KUKA KRL program: EPS_2_25694_RR01_A_20260120031656.src

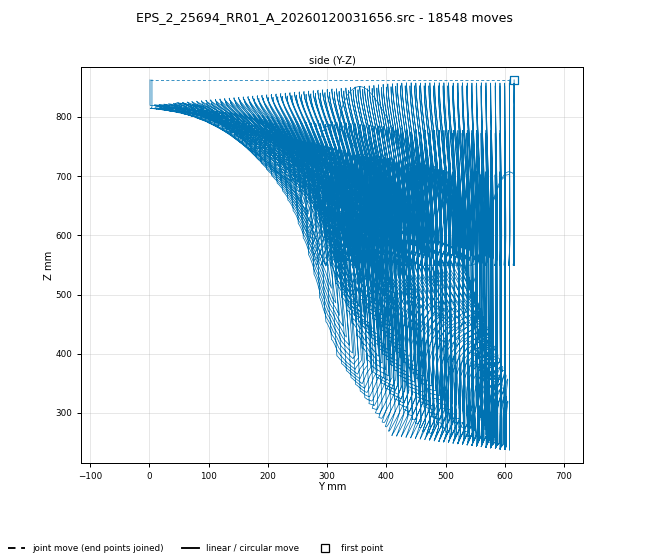
[picture p0: tool path of EPS_2_25694_RR01_A_20260120031656.src, 18548 of 18550 moves have a stored position in this frame; points joined in program order, loops and branches not executed]
&ACCESS RVP
&REL 4
&COMMENT QRS 19112012
&PARAM EDITMASK = *
DEF PART()
EXT BAS (BAS_COMMAND :IN,REAL :IN )
INT I
BAS (#INITMOV,0 )

;KUKA QRS Post kuka4.cps  Date:22-06-2017 !

File_ID=2993

QRS_PRE_INIT()

;Init var - Until changes are made in qrs_pre_init
Outlet_Square_prg=0
Inlet_1_Square_prg=0
Inlet_2_Square_prg=0
Inlet_3_Square_prg=0
Inlet_4_Square_prg=0
Inlet_5_Square_prg=0

Outlet_1={X 0.000, Y 425.000, Z 586.000, B 0.000, E1 0.000 }
Inlet_1={X 0.000, Y 537.740, Z 427.000, B 0.000, E1 94.000 }
Inlet_2={X 0.000, Y 466.000, Z 544.000, B 0.000, E1 177.000 }
Inlet_3={X 0.000, Y 531.490, Z 452.000, B 0.000, E1 275.000 }
Outlet_1_type=533
Inlet_1_type=201
Inlet_2_type=457
Inlet_3_type=251
;QRS#1=Sidecore dimensions
;QRS#2=525-21" Concrete
;QRS#3=200-8" PVC SDR 35
;QRS#4=450-18" Concrete
;QRS#5=250-10" PVC SDR 35
;QRS#6=
;QRS#7=
;QRS#8=
;QRS#9=S306-32
;QRS#10=12-08 PSX
;QRS#11=28A PSX-2
;QRS#12=14M PSX
;QRS#13=
;QRS#14=
;QRS#15=
;QRS#16=1220x127x1219 4'
;QRS#17=EPS Height
;QRS#18=852,5
;QRS#19=*
;QRS#20= UPDATED VERSION 22-06-2017
;QRS#21=*
Outlet_Square=0250
Inlet_1_Square=0100
Inlet_2_Square=0250
Inlet_3_Square=0100
Inlet_4_Square=0
Inlet_5_Square=0
Mill_Square=1
Outlet_Square_Prg=263
Inlet_1_Square_prg=204
Inlet_2_Square_prg=274
Inlet_3_Square_prg=205

QRS_INIT()

$ADVANCE=5

; T1
PTP {E1 172.342,E2 172.342}
PTP {X 0,Y 615.793,A -85,B 0,C 180,E1 172.342,E2 172.342,E3 0,E4 0,E5 0,E6 0}
QRS_SPEED_INIT()
LIN {X 0,Y 615.793,Z 862.5,A -85,B 0,C 180,E1 172.342,E2 172.342,E3 0,E4 0,E5 0,E6 0} C_VEL
LIN {X 0,Y 615.793,Z 711.666,A -85,B 0,C 180,E1 172.342,E2 172.342} C_VEL
LIN {X 0,Y 615.793,Z 703.764,A -85,B 0,C 180,E1 172.342,E2 172.342} C_VEL
LIN {X 0,Y 615.77,Z 701.828,A -85,B 0,C 180,E1 172.575,E2 172.575} C_VEL
LIN {X 0,Y 615.76,Z 703.691,A -85,B 0,C 180,E1 173.245,E2 173.245} C_VEL
LIN {X 0,Y 615.844,Z 705.541,A -85,B 0,C 180,E1 174.193,E2 174.193} C_VEL
LIN {X 0,Y 615.719,Z 706.621,A -85,B 0,C 180,E1 175.124,E2 175.124} C_VEL
LIN {X 0,Y 615.715,Z 706.871,A -85,B 0,C 180,E1 175.589,E2 175.589} C_VEL
LIN {X 0,Y 615.813,Z 706.79,A -85,B 0,C 180,E1 176.52,E2 176.52} C_VEL
LIN {X 0,Y 615.76,Z 705.947,A -85,B 0,C 180,E1 177.448,E2 177.448} C_VEL
LIN {X 0,Y 615.722,Z 704.334,A -85,B 0,C 180,E1 178.376,E2 178.376} C_VEL
LIN {X 0,Y 615.846,Z 701.911,A -85,B 0,C 180,E1 179.304,E2 179.304} C_VEL
LIN {X 0,Y 615.823,Z 700.411,A -85,B 0,C 180,E1 179.768,E2 179.768} C_VEL
LIN {X 0,Y 615.774,Z 698.687,A -85,B 0,C 180,E1 180.232,E2 180.232} C_VEL
LIN {X 0,Y 615.76,Z 695.634,A -85,B 0,C 180,E1 180.928,E2 180.928} C_VEL
LIN {X 0,Y 615.848,Z 692.021,A -85,B 0,C 180,E1 181.623,E2 181.623} C_VEL
LIN {X 0,Y 615.81,Z 687.854,A -85,B 0,C 180,E1 182.319,E2 182.319} C_VEL
LIN {X 0,Y 615.8,Z 682.955,A -85,B 0,C 180,E1 183.016,E2 183.016} C_VEL
LIN {X 0,Y 615.841,Z 677.301,A -85,B 0,C 180,E1 183.713,E2 183.713} C_VEL
LIN {X 0,Y 615.831,Z 671.884,A -85,B 0,C 180,E1 184.294,E2 184.294} C_VEL
LIN {X 0,Y 615.826,Z 665.734,A -85,B 0,C 180,E1 184.875,E2 184.875} C_VEL
LIN {X 0,Y 615.847,Z 658.636,A -85,B 0,C 180,E1 185.457,E2 185.457} C_VEL
LIN {X 0,Y 615.854,Z 652.201,A -85,B 0,C 180,E1 185.918,E2 185.918} C_VEL
LIN {X 0,Y 615.823,Z 645.096,A -85,B 0,C 180,E1 186.362,E2 186.362} C_VEL
LIN {X 0,Y 615.837,Z 636.811,A -85,B 0,C 180,E1 186.805,E2 186.805} C_VEL
LIN {X 0,Y 615.843,Z 629.456,A -85,B 0,C 180,E1 187.138,E2 187.138} C_VEL
LIN {X 0,Y 615.852,Z 620.279,A -85,B 0,C 180,E1 187.484,E2 187.484} C_VEL
LIN {X 0,Y 615.848,Z 611.384,A -85,B 0,C 180,E1 187.748,E2 187.748} C_VEL
LIN {X 0,Y 615.849,Z 602.82,A -85,B 0,C 180,E1 187.941,E2 187.941} C_VEL
LIN {X 0,Y 615.85,Z 593.381,A -85,B 0,C 180,E1 188.09,E2 188.09} C_VEL
LIN {X 0,Y 615.685,Z 559.528,A -85,B 0,C 180,E1 188.49,E2 188.49} C_VEL
LIN {X 0,Y 615.331,Z 549.53,A -85,B 0,C 180,E1 188.614,E2 188.614} C_VEL
LIN {X 0,Y 615.64,Z 549.53,A -85,B 0,C 180,E1 188.676,E2 188.676} C_VEL
LIN {X 0,Y 615.827,Z 549.53,A -85,B 0,C 180,E1 189.302,E2 189.302} C_VEL
LIN {X 0,Y 615.855,Z 549.53,A -85,B 0,C 180,E1 190.493,E2 190.493} C_VEL
LIN {X 0,Y 615.807,Z 549.53,A -85,B 0,C 180,E1 195.252,E2 195.252} C_VEL
LIN {X 0,Y 615.774,Z 549.53,A -85,B 0,C 180,E1 200.122,E2 200.122} C_VEL
LIN {X 0,Y 615.735,Z 549.53,A -85,B 0,C 180,E1 205.151,E2 205.151} C_VEL
LIN {X 0,Y 615.403,Z 549.53,A -85,B 0,C 180,E1 209.459,E2 209.459} C_VEL
LIN {X 0,Y 615.737,Z 549.53,A -85,B 0,C 180,E1 210.395,E2 210.395} C_VEL
LIN {X 0,Y 615.132,Z 549.53,A -85,B 0,C 180,E1 213.842,E2 213.842} C_VEL
LIN {X 0,Y 615.665,Z 549.53,A -85,B 0,C 180,E1 215.943,E2 215.943} C_VEL
LIN {X 0,Y 615.412,Z 549.53,A -85,B 0,C 180,E1 217.842,E2 217.842} C_VEL
LIN {X 0,Y 615.369,Z 549.53,A -85,B 0,C 180,E1 218.885,E2 218.885} C_VEL
LIN {X 0,Y 615.653,Z 549.53,A -85,B 0,C 180,E1 221.504,E2 221.504} C_VEL
LIN {X 0,Y 615.675,Z 549.53,A -85,B 0,C 180,E1 225.105,E2 225.105} C_VEL
LIN {X 0,Y 615.271,Z 549.53,A -85,B 0,C 180,E1 228.537,E2 228.537} C_VEL
LIN {X 0,Y 615.658,Z 549.53,A -85,B 0,C 180,E1 231.137,E2 231.137} C_VEL
LIN {X 0,Y 615.637,Z 549.53,A -85,B 0,C 180,E1 236.088,E2 236.088} C_VEL
LIN {X 0,Y 615.75,Z 549.53,A -85,B 0,C 180,E1 236.878,E2 236.878} C_VEL
LIN {X 0,Y 615.843,Z 549.53,A -85,B 0,C 180,E1 240.621,E2 240.621} C_VEL
LIN {X 0,Y 615.218,Z 549.53,A -85,B 0,C 180,E1 240.78,E2 240.78} C_VEL
LIN {X 0,Y 615.11,Z 550.038,A -85,B 0,C 180,E1 240.802,E2 240.802} C_VEL
LIN {X 0,Y 615.44,Z 600.029,A -85,B 0,C 180,E1 241.477,E2 241.477} C_VEL
LIN {X 0,Y 615.51,Z 611.094,A -85,B 0,C 180,E1 241.655,E2 241.655} C_VEL
LIN {X 0,Y 615.537,Z 625.6,A -85,B 0,C 180,E1 241.961,E2 241.961} C_VEL
LIN {X 0,Y 615.51,Z 635.908,A -85,B 0,C 180,E1 242.221,E2 242.221} C_VEL
LIN {X 0,Y 615.677,Z 651.509,A -85,B 0,C 180,E1 242.705,E2 242.705} C_VEL
LIN {X 0,Y 615.645,Z 663.945,A -85,B 0,C 180,E1 243.152,E2 243.152} C_VEL
LIN {X 0,Y 615.577,Z 673.861,A -85,B 0,C 180,E1 243.554,E2 243.554} C_VEL
LIN {X 0,Y 615.711,Z 689.587,A -85,B 0,C 180,E1 244.286,E2 244.286} C_VEL
LIN {X 0,Y 615.692,Z 701.936,A -85,B 0,C 180,E1 244.935,E2 244.935} C_VEL
LIN {X 0,Y 615.677,Z 713.616,A -85,B 0,C 180,E1 245.617,E2 245.617} C_VEL
LIN {X 0,Y 615.714,Z 725.406,A -85,B 0,C 180,E1 246.38,E2 246.38} C_VEL
LIN {X 0,Y 615.721,Z 736.083,A -85,B 0,C 180,E1 247.135,E2 247.135} C_VEL
LIN {X 0,Y 615.707,Z 747.387,A -85,B 0,C 180,E1 248.011,E2 248.011} C_VEL
LIN {X 0,Y 615.704,Z 756.649,A -85,B 0,C 180,E1 248.791,E2 248.791} C_VEL
LIN {X 0,Y 615.752,Z 766.786,A -85,B 0,C 180,E1 249.722,E2 249.722} C_VEL
LIN {X 0,Y 615.723,Z 776.05,A -85,B 0,C 180,E1 250.646,E2 250.646} C_VEL
LIN {X 0,Y 615.683,Z 784.412,A -85,B 0,C 180,E1 251.548,E2 251.548} C_VEL
LIN {X 0,Y 615.766,Z 792.772,A -85,B 0,C 180,E1 252.531,E2 252.531} C_VEL
LIN {X 0,Y 615.718,Z 800.678,A -85,B 0,C 180,E1 253.541,E2 253.541} C_VEL
LIN {X 0,Y 615.581,Z 807.424,A -85,B 0,C 180,E1 254.472,E2 254.472} C_VEL
LIN {X 0,Y 615.671,Z 815.058,A -85,B 0,C 180,E1 255.644,E2 255.644} C_VEL
LIN {X 0,Y 615.807,Z 820.435,A -85,B 0,C 180,E1 256.543,E2 256.543} C_VEL
LIN {X 0,Y 615.575,Z 826.908,A -85,B 0,C 180,E1 257.728,E2 257.728} C_VEL
LIN {X 0,Y 615.615,Z 832.623,A -85,B 0,C 180,E1 258.913,E2 258.913} C_VEL
LIN {X 0,Y 615.829,Z 837.633,A -85,B 0,C 180,E1 260.096,E2 260.096} C_VEL
LIN {X 0,Y 615.604,Z 842.062,A -85,B 0,C 180,E1 261.268,E2 261.268} C_VEL
LIN {X 0,Y 615.654,Z 846.465,A -85,B 0,C 180,E1 262.658,E2 262.658} C_VEL
LIN {X 0,Y 615.788,Z 849.368,A -85,B 0,C 180,E1 263.748,E2 263.748} C_VEL
LIN {X 0,Y 615.542,Z 852.381,A -85,B 0,C 180,E1 265.122,E2 265.122} C_VEL
LIN {X 0,Y 615.642,Z 854.591,A -85,B 0,C 180,E1 266.519,E2 266.519} C_VEL
LIN {X 0,Y 615.712,Z 856.054,A -85,B 0,C 180,E1 267.912,E2 267.912} C_VEL
LIN {X 0,Y 615.553,Z 856.715,A -85,B 0,C 180,E1 268.84,E2 268.84} C_VEL
LIN {X 0,Y 615.842,Z 856.659,A -85,B 0,C 180,E1 271.159,E2 271.159} C_VEL
LIN {X 0,Y 615.631,Z 856.069,A -85,B 0,C 180,E1 272.088,E2 272.088} C_VEL
LIN {X 0,Y 615.55,Z 854.608,A -85,B 0,C 180,E1 273.482,E2 273.482} C_VEL
LIN {X 0,Y 615.828,Z 852.329,A -85,B 0,C 180,E1 274.875,E2 274.875} C_VEL
LIN {X 0,Y 615.615,Z 849.404,A -85,B 0,C 180,E1 276.251,E2 276.251} C_VEL
LIN {X 0,Y 615.622,Z 846.266,A -85,B 0,C 180,E1 277.418,E2 277.418} C_VEL
LIN {X 0,Y 615.784,Z 842.035,A -85,B 0,C 180,E1 278.73,E2 278.73} C_VEL
LIN {X 0,Y 615.572,Z 837.67,A -85,B 0,C 180,E1 279.908,E2 279.908} C_VEL
LIN {X 0,Y 615.632,Z 832.621,A -85,B 0,C 180,E1 281.087,E2 281.087} C_VEL
LIN {X 0,Y 615.805,Z 826.881,A -85,B 0,C 180,E1 282.267,E2 282.267} C_VEL
LIN {X 0,Y 615.626,Z 820.453,A -85,B 0,C 180,E1 283.461,E2 283.461} C_VEL
LIN {X 0,Y 615.698,Z 813.192,A -85,B 0,C 180,E1 284.655,E2 284.655} C_VEL
LIN {X 0,Y 615.811,Z 807.63,A -85,B 0,C 180,E1 285.489,E2 285.489} C_VEL
LIN {X 0,Y 615.663,Z 798.196,A -85,B 0,C 180,E1 286.791,E2 286.791} C_VEL
LIN {X 0,Y 615.737,Z 789.604,A -85,B 0,C 180,E1 287.853,E2 287.853} C_VEL
LIN {X 0,Y 615.77,Z 781.409,A -85,B 0,C 180,E1 288.785,E2 288.785} C_VEL
LIN {X 0,Y 615.697,Z 771.52,A -85,B 0,C 180,E1 289.817,E2 289.817} C_VEL
LIN {X 0,Y 615.715,Z 763.533,A -85,B 0,C 180,E1 290.588,E2 290.588} C_VEL
LIN {X 0,Y 615.746,Z 753.03,A -85,B 0,C 180,E1 291.519,E2 291.519} C_VEL
LIN {X 0,Y 615.704,Z 743.049,A -85,B 0,C 180,E1 292.335,E2 292.335} C_VEL
LIN {X 0,Y 615.702,Z 733.289,A -85,B 0,C 180,E1 293.072,E2 293.072} C_VEL
LIN {X 0,Y 615.683,Z 721.63,A -85,B 0,C 180,E1 293.874,E2 293.874} C_VEL
LIN {X 0,Y 615.688,Z 709.594,A -85,B 0,C 180,E1 294.624,E2 294.624} C_VEL
LIN {X 0,Y 615.65,Z 698.88,A -85,B 0,C 180,E1 295.235,E2 295.235} C_VEL
LIN {X 0,Y 615.644,Z 688.01,A -85,B 0,C 180,E1 295.797,E2 295.797} C_VEL
LIN {X 0,Y 615.702,Z 673.863,A -85,B 0,C 180,E1 296.44,E2 296.44} C_VEL
LIN {X 0,Y 615.617,Z 660.66,A -85,B 0,C 180,E1 296.972,E2 296.972} C_VEL
LIN {X 0,Y 615.561,Z 651.512,A -85,B 0,C 180,E1 297.3,E2 297.3} C_VEL
LIN {X 0,Y 615.623,Z 634.838,A -85,B 0,C 180,E1 297.801,E2 297.801} C_VEL
LIN {X 0,Y 615.442,Z 622.423,A -85,B 0,C 180,E1 298.118,E2 298.118} C_VEL
LIN {X 0,Y 615.592,Z 610.944,A -85,B 0,C 180,E1 298.344,E2 298.344} C_VEL
LIN {X 0,Y 615.568,Z 593.456,A -85,B 0,C 180,E1 298.608,E2 298.608} C_VEL
LIN {X 0,Y 615.164,Z 549.53,A -85,B 0,C 180,E1 299.213,E2 299.213} C_VEL
LIN {X 0,Y 615.78,Z 549.53,A -85,B 0,C 180,E1 299.347,E2 299.347} C_VEL
LIN {X 0,Y 615.858,Z 549.53,A -85,B 0,C 180,E1 300.388,E2 300.388} C_VEL
LIN {X 0,Y 615.152,Z 549.53,A -85,B 0,C 180,E1 303.844,E2 303.844} C_VEL
LIN {X 0,Y 615.699,Z 549.53,A -85,B 0,C 180,E1 305.94,E2 305.94} C_VEL
LIN {X 0,Y 615.75,Z 549.53,A -85,B 0,C 180,E1 308.856,E2 308.856} C_VEL
LIN {X 0,Y 615.251,Z 549.53,A -85,B 0,C 180,E1 311.943,E2 311.943} C_VEL
LIN {X 0,Y 615.68,Z 549.53,A -85,B 0,C 180,E1 314.895,E2 314.895} C_VEL
LIN {X 0,Y 615.655,Z 549.53,A -85,B 0,C 180,E1 318.496,E2 318.496} C_VEL
LIN {X 0,Y 615.378,Z 549.53,A -85,B 0,C 180,E1 321.116,E2 321.116} C_VEL
LIN {X 0,Y 615.434,Z 549.53,A -85,B 0,C 180,E1 322.155,E2 322.155} C_VEL
LIN {X 0,Y 615.69,Z 549.53,A -85,B 0,C 180,E1 324.059,E2 324.059} C_VEL
LIN {X 0,Y 615.15,Z 549.53,A -85,B 0,C 180,E1 326.842,E2 326.842} C_VEL
LIN {X 0,Y 615.741,Z 549.53,A -85,B 0,C 180,E1 329.606,E2 329.606} C_VEL
LIN {X 0,Y 615.23,Z 549.53,A -85,B 0,C 180,E1 332.234,E2 332.234} C_VEL
LIN {X 0,Y 615.761,Z 549.53,A -85,B 0,C 180,E1 334.85,E2 334.85} C_VEL
LIN {X 0,Y 615.815,Z 549.53,A -85,B 0,C 180,E1 339.879,E2 339.879} C_VEL
LIN {X 0,Y 615.435,Z 549.53,A -85,B 0,C 180,E1 340.175,E2 340.175} C_VEL
LIN {X 0,Y 615.817,Z 577.641,A -85,B 0,C 180,E1 340.534,E2 340.534} C_VEL
LIN {X 0,Y 615.772,Z 587.447,A -85,B 0,C 180,E1 340.724,E2 340.724} C_VEL
LIN {X 0,Y 615.854,Z 596.495,A -85,B 0,C 180,E1 340.957,E2 340.957} C_VEL
LIN {X 0,Y 615.859,Z 606.239,A -85,B 0,C 180,E1 341.268,E2 341.268} C_VEL
LIN {X 0,Y 615.823,Z 614.32,A -85,B 0,C 180,E1 341.582,E2 341.582} C_VEL
LIN {X 0,Y 615.846,Z 622.438,A -85,B 0,C 180,E1 341.95,E2 341.95} C_VEL
LIN {X 0,Y 615.84,Z 631.644,A -85,B 0,C 180,E1 342.432,E2 342.432} C_VEL
LIN {X 0,Y 615.814,Z 639.845,A -85,B 0,C 180,E1 342.935,E2 342.935} C_VEL
LIN {X 0,Y 615.812,Z 647.097,A -85,B 0,C 180,E1 343.438,E2 343.438} C_VEL
LIN {X 0,Y 615.784,Z 654.157,A -85,B 0,C 180,E1 343.988,E2 343.988} C_VEL
LIN {X 0,Y 615.838,Z 661.067,A -85,B 0,C 180,E1 344.603,E2 344.603} C_VEL
LIN {X 0,Y 615.825,Z 667.082,A -85,B 0,C 180,E1 345.199,E2 345.199} C_VEL
LIN {X 0,Y 615.781,Z 673.744,A -85,B 0,C 180,E1 345.946,E2 345.946} C_VEL
LIN {X 0,Y 615.829,Z 679.56,A -85,B 0,C 180,E1 346.693,E2 346.693} C_VEL
LIN {X 0,Y 615.806,Z 684.677,A -85,B 0,C 180,E1 347.436,E2 347.436} C_VEL
LIN {X 0,Y 615.751,Z 688.277,A -85,B 0,C 180,E1 348.028,E2 348.028} C_VEL
LIN {X 0,Y 615.762,Z 691.495,A -85,B 0,C 180,E1 348.62,E2 348.62} C_VEL
LIN {X 0,Y 615.825,Z 694.353,A -85,B 0,C 180,E1 349.212,E2 349.212} C_VEL
LIN {X 0,Y 615.751,Z 698.006,A -85,B 0,C 180,E1 350.095,E2 350.095} C_VEL
LIN {X 0,Y 615.714,Z 700.083,A -85,B 0,C 180,E1 350.682,E2 350.682} C_VEL
LIN {X 0,Y 615.74,Z 701.861,A -85,B 0,C 180,E1 351.27,E2 351.27} C_VEL
LIN {X 0,Y 615.83,Z 703.353,A -85,B 0,C 180,E1 351.857,E2 351.857} C_VEL
LIN {X 0,Y 615.793,Z 704.79,A -85,B 0,C 180,E1 352.558,E2 352.558} C_VEL
LIN {X 0,Y 615.725,Z 705.932,A -85,B 0,C 180,E1 353.321,E2 353.321} C_VEL
LIN {X 0,Y 615.786,Z 706.705,A -85,B 0,C 180,E1 354.193,E2 354.193} C_VEL
LIN {X 0,Y 615.837,Z 706.863,A -85,B 0,C 180,E1 354.659,E2 354.659} C_VEL
LIN {X 0,Y 615.739,Z 706.797,A -85,B 0,C 180,E1 355.589,E2 355.589} C_VEL
LIN {X 0,Y 615.737,Z 706.013,A -85,B 0,C 180,E1 356.519,E2 356.519} C_VEL
LIN {X 0,Y 615.848,Z 704.619,A -85,B 0,C 180,E1 357.449,E2 357.449} C_VEL
LIN {X 0,Y 615.726,Z 702.572,A -85,B 0,C 180,E1 358.376,E2 358.376} C_VEL
LIN {X 0,Y 615.717,Z 701.319,A -85,B 0,C 180,E1 358.84,E2 358.84} C_VEL
LIN {X 0,Y 615.818,Z 698.168,A -85,B 0,C 180,E1 359.768,E2 359.768} C_VEL
LIN {X 0,Y 615.764,Z 694.376,A -85,B 0,C 180,E1 360.696,E2 360.696} C_VEL
LIN {X 0,Y 615.727,Z 689.697,A -85,B 0,C 180,E1 361.624,E2 361.624} C_VEL
LIN {X 0,Y 615.85,Z 684.163,A -85,B 0,C 180,E1 362.551,E2 362.551} C_VEL
LIN {X 0,Y 615.793,Z 679.339,A -85,B 0,C 180,E1 363.248,E2 363.248} C_VEL
LIN {X 0,Y 615.754,Z 673.904,A -85,B 0,C 180,E1 363.946,E2 363.946} C_VEL
LIN {X 0,Y 615.827,Z 667.753,A -85,B 0,C 180,E1 364.643,E2 364.643} C_VEL
LIN {X 0,Y 615.83,Z 660.706,A -85,B 0,C 180,E1 365.341,E2 365.341} C_VEL
LIN {X 0,Y 615.808,Z 654.083,A -85,B 0,C 180,E1 365.927,E2 365.927} C_VEL
LIN {X 0,Y 615.834,Z 646.301,A -85,B 0,C 180,E1 366.529,E2 366.529} C_VEL
LIN {X 0,Y 615.833,Z 639.954,A -85,B 0,C 180,E1 366.967,E2 366.967} C_VEL
LIN {X 0,Y 615.822,Z 631.782,A -85,B 0,C 180,E1 367.47,E2 367.47} C_VEL
LIN {X 0,Y 615.822,Z 623.205,A -85,B 0,C 180,E1 367.924,E2 367.924} C_VEL
LIN {X 0,Y 615.787,Z 616.943,A -85,B 0,C 180,E1 368.217,E2 368.217} C_VEL
LIN {X 0,Y 615.839,Z 609.792,A -85,B 0,C 180,E1 368.509,E2 368.509} C_VEL
LIN {X 0,Y 615.83,Z 601.453,A -85,B 0,C 180,E1 368.802,E2 368.802} C_VEL
LIN {X 0,Y 615.816,Z 592.021,A -85,B 0,C 180,E1 369.078,E2 369.078} C_VEL
LIN {X 0,Y 615.861,Z 581.948,A -85,B 0,C 180,E1 369.297,E2 369.297} C_VEL
LIN {X 0,Y 615.867,Z 573.067,A -85,B 0,C 180,E1 369.44,E2 369.44} C_VEL
LIN {X 0,Y 615.676,Z 558.016,A -85,B 0,C 180,E1 369.626,E2 369.626} C_VEL
LIN {X 0,Y 614.954,Z 549.53,A -85,B 0,C 180,E1 369.744,E2 369.744} C_VEL
LIN {X 0,Y 615.72,Z 549.53,A -85,B 0,C 180,E1 369.885,E2 369.885} C_VEL
LIN {X 0,Y 615.756,Z 549.53,A -85,B 0,C 180,E1 370.494,E2 370.494} C_VEL
LIN {X 0,Y 615.824,Z 549.53,A -85,B 0,C 180,E1 372.861,E2 372.861} C_VEL
LIN {X 0,Y 615.82,Z 549.53,A -85,B 0,C 180,E1 377.67,E2 377.67} C_VEL
LIN {X 0,Y 615.819,Z 549.53,A -85,B 0,C 180,E1 377.999,E2 377.999} C_VEL
LIN {X 0,Y 615.769,Z 549.53,A -85,B 0,C 180,E1 382.613,E2 382.613} C_VEL
LIN {X 0,Y 615.234,Z 549.53,A -85,B 0,C 180,E1 385.173,E2 385.173} C_VEL
LIN {X 0,Y 615.747,Z 549.53,A -85,B 0,C 180,E1 387.741,E2 387.741} C_VEL
LIN {X 0,Y 615.173,Z 549.53,A -85,B 0,C 180,E1 390.425,E2 390.425} C_VEL
LIN {X 0,Y 615.698,Z 549.53,A -85,B 0,C 180,E1 393.125,E2 393.125} C_VEL
LIN {X 0,Y 615.641,Z 549.53,A -85,B 0,C 180,E1 393.912,E2 393.912} C_VEL
LIN {X 0,Y 615.65,Z 549.53,A -85,B 0,C 180,E1 398.864,E2 398.864} C_VEL
LIN {X 0,Y 615.251,Z 549.53,A -85,B 0,C 180,E1 401.943,E2 401.943} C_VEL
LIN {X 0,Y 615.677,Z 549.53,A -85,B 0,C 180,E1 404.895,E2 404.895} C_VEL
LIN {X 0,Y 615.656,Z 549.53,A -85,B 0,C 180,E1 408.496,E2 408.496} C_VEL
LIN {X 0,Y 615.364,Z 549.53,A -85,B 0,C 180,E1 411.115,E2 411.115} C_VEL
LIN {X 0,Y 615.411,Z 549.53,A -85,B 0,C 180,E1 412.158,E2 412.158} C_VEL
LIN {X 0,Y 615.666,Z 549.53,A -85,B 0,C 180,E1 414.058,E2 414.058} C_VEL
LIN {X 0,Y 615.12,Z 549.53,A -85,B 0,C 180,E1 416.84,E2 416.84} C_VEL
LIN {X 0,Y 615.705,Z 549.53,A -85,B 0,C 180,E1 419.604,E2 419.604} C_VEL
LIN {X 0,Y 615.214,Z 549.53,A -85,B 0,C 180,E1 422.233,E2 422.233} C_VEL
LIN {X 0,Y 615.802,Z 549.53,A -85,B 0,C 180,E1 424.852,E2 424.852} C_VEL
LIN {X 0,Y 615.794,Z 549.53,A -85,B 0,C 180,E1 427.802,E2 427.802} C_VEL
LIN {X 0,Y 615.45,Z 549.53,A -85,B 0,C 180,E1 428.294,E2 428.294} C_VEL
LIN {X 0,Y 615.732,Z 564.984,A -85,B 0,C 180,E1 428.558,E2 428.558} C_VEL
LIN {X 0,Y 615.758,Z 576.642,A -85,B 0,C 180,E1 428.802,E2 428.802} C_VEL
LIN {X 0,Y 615.661,Z 588.21,A -85,B 0,C 180,E1 429.097,E2 429.097} C_VEL
LIN {X 0,Y 615.664,Z 595.98,A -85,B 0,C 180,E1 429.326,E2 429.326} C_VEL
LIN {X 0,Y 615.747,Z 610.255,A -85,B 0,C 180,E1 429.831,E2 429.831} C_VEL
LIN {X 0,Y 615.696,Z 620.874,A -85,B 0,C 180,E1 430.26,E2 430.26} C_VEL
LIN {X 0,Y 615.723,Z 630.978,A -85,B 0,C 180,E1 430.723,E2 430.723} C_VEL
LIN {X 0,Y 615.744,Z 642.478,A -85,B 0,C 180,E1 431.316,E2 431.316} C_VEL
LIN {X 0,Y 615.692,Z 653.357,A -85,B 0,C 180,E1 431.941,E2 431.941} C_VEL
LIN {X 0,Y 615.75,Z 662.642,A -85,B 0,C 180,E1 432.531,E2 432.531} C_VEL
LIN {X 0,Y 615.751,Z 671.436,A -85,B 0,C 180,E1 433.139,E2 433.139} C_VEL
LIN {X 0,Y 615.773,Z 680.767,A -85,B 0,C 180,E1 433.845,E2 433.845} C_VEL
LIN {X 0,Y 615.759,Z 689.864,A -85,B 0,C 180,E1 434.597,E2 434.597} C_VEL
LIN {X 0,Y 615.723,Z 698.194,A -85,B 0,C 180,E1 435.346,E2 435.346} C_VEL
LIN {X 0,Y 615.752,Z 705.849,A -85,B 0,C 180,E1 436.095,E2 436.095} C_VEL
LIN {X 0,Y 615.781,Z 714.208,A -85,B 0,C 180,E1 436.989,E2 436.989} C_VEL
LIN {X 0,Y 615.693,Z 720.632,A -85,B 0,C 180,E1 437.73,E2 437.73} C_VEL
LIN {X 0,Y 615.688,Z 727.672,A -85,B 0,C 180,E1 438.619,E2 438.619} C_VEL
LIN {X 0,Y 615.803,Z 734.076,A -85,B 0,C 180,E1 439.507,E2 439.507} C_VEL
LIN {X 0,Y 615.719,Z 739.937,A -85,B 0,C 180,E1 440.388,E2 440.388} C_VEL
LIN {X 0,Y 615.637,Z 745.266,A -85,B 0,C 180,E1 441.268,E2 441.268} C_VEL
LIN {X 0,Y 615.758,Z 751.733,A -85,B 0,C 180,E1 442.482,E2 442.482} C_VEL
LIN {X 0,Y 615.733,Z 756.514,A -85,B 0,C 180,E1 443.487,E2 443.487} C_VEL
LIN {X 0,Y 615.621,Z 759.555,A -85,B 0,C 180,E1 444.191,E2 444.191} C_VEL
LIN {X 0,Y 615.66,Z 764.751,A -85,B 0,C 180,E1 445.589,E2 445.589} C_VEL
LIN {X 0,Y 615.831,Z 767.675,A -85,B 0,C 180,E1 446.52,E2 446.52} C_VEL
LIN {X 0,Y 615.654,Z 770.202,A -85,B 0,C 180,E1 447.448,E2 447.448} C_VEL
LIN {X 0,Y 615.615,Z 773.188,A -85,B 0,C 180,E1 448.84,E2 448.84} C_VEL
LIN {X 0,Y 615.79,Z 774.69,A -85,B 0,C 180,E1 449.768,E2 449.768} C_VEL
LIN {X 0,Y 615.612,Z 776.208,A -85,B 0,C 180,E1 451.16,E2 451.16} C_VEL
LIN {X 0,Y 615.593,Z 776.775,A -85,B 0,C 180,E1 452.088,E2 452.088} C_VEL
LIN {X 0,Y 615.82,Z 776.809,A -85,B 0,C 180,E1 453.48,E2 453.48} C_VEL
LIN {X 0,Y 615.671,Z 776.437,A -85,B 0,C 180,E1 454.411,E2 454.411} C_VEL
LIN {X 0,Y 615.674,Z 775.106,A -85,B 0,C 180,E1 455.808,E2 455.808} C_VEL
LIN {X 0,Y 615.821,Z 773.867,A -85,B 0,C 180,E1 456.639,E2 456.639} C_VEL
LIN {X 0,Y 615.694,Z 772.396,A -85,B 0,C 180,E1 457.473,E2 457.473} C_VEL
LIN {X 0,Y 615.627,Z 770.945,A -85,B 0,C 180,E1 458.146,E2 458.146} C_VEL
LIN {X 0,Y 615.712,Z 767.892,A -85,B 0,C 180,E1 459.318,E2 459.318} C_VEL
LIN {X 0,Y 615.824,Z 766.051,A -85,B 0,C 180,E1 459.904,E2 459.904} C_VEL
LIN {X 0,Y 615.691,Z 763.091,A -85,B 0,C 180,E1 460.79,E2 460.79} C_VEL
LIN {X 0,Y 615.621,Z 759.728,A -85,B 0,C 180,E1 461.679,E2 461.679} C_VEL
LIN {X 0,Y 615.698,Z 755.906,A -85,B 0,C 180,E1 462.567,E2 462.567} C_VEL
LIN {X 0,Y 615.808,Z 751.584,A -85,B 0,C 180,E1 463.457,E2 463.457} C_VEL
LIN {X 0,Y 615.654,Z 745.18,A -85,B 0,C 180,E1 464.656,E2 464.656} C_VEL
LIN {X 0,Y 615.723,Z 738.859,A -85,B 0,C 180,E1 465.689,E2 465.689} C_VEL
LIN {X 0,Y 615.783,Z 732.292,A -85,B 0,C 180,E1 466.659,E2 466.659} C_VEL
LIN {X 0,Y 615.658,Z 724.7,A -85,B 0,C 180,E1 467.675,E2 467.675} C_VEL
LIN {X 0,Y 615.689,Z 718.409,A -85,B 0,C 180,E1 468.444,E2 468.444} C_VEL
LIN {X 0,Y 615.801,Z 710.262,A -85,B 0,C 180,E1 469.352,E2 469.352} C_VEL
LIN {X 0,Y 615.747,Z 702.76,A -85,B 0,C 180,E1 470.123,E2 470.123} C_VEL
LIN {X 0,Y 615.733,Z 694.557,A -85,B 0,C 180,E1 470.898,E2 470.898} C_VEL
LIN {X 0,Y 615.764,Z 685.562,A -85,B 0,C 180,E1 471.674,E2 471.674} C_VEL
LIN {X 0,Y 615.766,Z 677.142,A -85,B 0,C 180,E1 472.345,E2 472.345} C_VEL
LIN {X 0,Y 615.749,Z 668.827,A -85,B 0,C 180,E1 472.957,E2 472.957} C_VEL
LIN {X 0,Y 615.745,Z 658.529,A -85,B 0,C 180,E1 473.647,E2 473.647} C_VEL
LIN {X 0,Y 615.736,Z 649.08,A -85,B 0,C 180,E1 474.223,E2 474.223} C_VEL
LIN {X 0,Y 615.756,Z 638.597,A -85,B 0,C 180,E1 474.801,E2 474.801} C_VEL
LIN {X 0,Y 615.711,Z 628.358,A -85,B 0,C 180,E1 475.312,E2 475.312} C_VEL
LIN {X 0,Y 615.667,Z 619.423,A -85,B 0,C 180,E1 475.716,E2 475.716} C_VEL
LIN {X 0,Y 615.75,Z 606.064,A -85,B 0,C 180,E1 476.236,E2 476.236} C_VEL
LIN {X 0,Y 615.692,Z 593.924,A -85,B 0,C 180,E1 476.643,E2 476.643} C_VEL
LIN {X 0,Y 615.602,Z 584.073,A -85,B 0,C 180,E1 476.932,E2 476.932} C_VEL
LIN {X 0,Y 615.713,Z 572.185,A -85,B 0,C 180,E1 477.211,E2 477.211} C_VEL
LIN {X 0,Y 615.625,Z 558.958,A -85,B 0,C 180,E1 477.46,E2 477.46} C_VEL
LIN {X 0,Y 615.415,Z 553.734,A -85,B 0,C 180,E1 477.547,E2 477.547} C_VEL
LIN {X 0,Y 614.53,Z 550.211,A -85,B 0,C 180,E1 477.636,E2 477.636} C_VEL
LIN {X 0,Y 614.522,Z 549.53,A -85,B 0,C 180,E1 477.678,E2 477.678} C_VEL
LIN {X 0,Y 615.217,Z 549.53,A -85,B 0,C 180,E1 477.767,E2 477.767} C_VEL
LIN {X 0,Y 615.367,Z 549.53,A -85,B 0,C 180,E1 479.453,E2 479.453} C_VEL
LIN {X 0,Y 615.847,Z 549.53,A -85,B 0,C 180,E1 483.116,E2 483.116} C_VEL
LIN {X 0,Y 615.539,Z 549.53,A -85,B 0,C 180,E1 485.951,E2 485.951} C_VEL
LIN {X 0,Y 615.605,Z 549.53,A -85,B 0,C 180,E1 487.865,E2 487.865} C_VEL
LIN {X 0,Y 615.661,Z 549.53,A -85,B 0,C 180,E1 491.908,E2 491.908} C_VEL
LIN {X 0,Y 615.214,Z 549.53,A -85,B 0,C 180,E1 495.148,E2 495.148} C_VEL
LIN {X 0,Y 615.68,Z 549.53,A -85,B 0,C 180,E1 498.093,E2 498.093} C_VEL
LIN {X 0,Y 615.608,Z 549.53,A -85,B 0,C 180,E1 502.134,E2 502.134} C_VEL
LIN {X 0,Y 615.572,Z 549.53,A -85,B 0,C 180,E1 504.051,E2 504.051} C_VEL
LIN {X 0,Y 615.72,Z 549.53,A -85,B 0,C 180,E1 506.077,E2 506.077} C_VEL
LIN {X 0,Y 615.716,Z 549.53,A -85,B 0,C 180,E1 506.876,E2 506.876} C_VEL
LIN {X 0,Y 615.549,Z 549.53,A -85,B 0,C 180,E1 510.517,E2 510.517} C_VEL
LIN {X 0,Y 615.49,Z 549.53,A -85,B 0,C 180,E1 512.247,E2 512.247} C_VEL
LIN {X 0,Y 615.283,Z 549.53,A -85,B 0,C 180,E1 515.698,E2 515.698} C_VEL
LIN {X 0,Y 615.753,Z 549.53,A -85,B 0,C 180,E1 517.386,E2 517.386} C_VEL
LIN {X 0,Y 615.811,Z 549.53,A -85,B 0,C 180,E1 522.808,E2 522.808} C_VEL
LIN {X 0,Y 615.751,Z 549.53,A -85,B 0,C 180,E1 523.017,E2 523.017} C_VEL
LIN {X 0,Y 614.742,Z 549.53,A -85,B 0,C 180,E1 523.199,E2 523.199} C_VEL
LIN {X 0,Y 613.931,Z 549.53,A -85,B 0,C 180,E1 523.262,E2 523.262} C_VEL
LIN {X 0,Y 615.12,Z 555.991,A -85,B 0,C 180,E1 523.367,E2 523.367} C_VEL
LIN {X 0,Y 615.778,Z 563.786,A -85,B 0,C 180,E1 523.472,E2 523.472} C_VEL
LIN {X 0,Y 615.845,Z 597.209,A -85,B 0,C 180,E1 523.873,E2 523.873} C_VEL
LIN {X 0,Y 615.865,Z 606.642,A -85,B 0,C 180,E1 524.049,E2 524.049} C_VEL
LIN {X 0,Y 615.82,Z 615.286,A -85,B 0,C 180,E1 524.268,E2 524.268} C_VEL
LIN {X 0,Y 615.821,Z 623.627,A -85,B 0,C 180,E1 524.543,E2 524.543} C_VEL
LIN {X 0,Y 615.824,Z 630.689,A -85,B 0,C 180,E1 524.823,E2 524.823} C_VEL
LIN {X 0,Y 615.828,Z 638.718,A -85,B 0,C 180,E1 525.199,E2 525.199} C_VEL
LIN {X 0,Y 615.828,Z 646.778,A -85,B 0,C 180,E1 525.648,E2 525.648} C_VEL
LIN {X 0,Y 615.812,Z 654.787,A -85,B 0,C 180,E1 526.17,E2 526.17} C_VEL
LIN {X 0,Y 615.822,Z 661.698,A -85,B 0,C 180,E1 526.693,E2 526.693} C_VEL
LIN {X 0,Y 615.846,Z 668.498,A -85,B 0,C 180,E1 527.288,E2 527.288} C_VEL
LIN {X 0,Y 615.805,Z 674.466,A -85,B 0,C 180,E1 527.881,E2 527.881} C_VEL
LIN {X 0,Y 615.772,Z 679.638,A -85,B 0,C 180,E1 528.472,E2 528.472} C_VEL
LIN {X 0,Y 615.848,Z 685.288,A -85,B 0,C 180,E1 529.212,E2 529.212} C_VEL
LIN {X 0,Y 615.781,Z 690.969,A -85,B 0,C 180,E1 530.095,E2 530.095} C_VEL
LIN {X 0,Y 615.745,Z 694.175,A -85,B 0,C 180,E1 530.683,E2 530.683} C_VEL
LIN {X 0,Y 615.833,Z 698.202,A -85,B 0,C 180,E1 531.564,E2 531.564} C_VEL
LIN {X 0,Y 615.818,Z 700.486,A -85,B 0,C 180,E1 532.163,E2 532.163} C_VEL
LIN {X 0,Y 615.77,Z 701.828,A -85,B 0,C 180,E1 532.575,E2 532.575} C_VEL
LIN {X 0,Y 613.247,Z 705.176,A -85,B 0,C 180,E1 533.744,E2 533.744} C_VEL
LIN {X 0,Y 607.956,Z 707.497,A -85,B 0,C 180,E1 535.521,E2 535.521} C_VEL
LIN {X 0,Y 607.848,Z 707.453,A -85,B 0,C 180,E1 535.728,E2 535.728} C_VEL
LIN {X 0,Y 607.862,Z 705.896,A -85,B 0,C 180,E1 537.863,E2 537.863} C_VEL
LIN {X 0,Y 607.909,Z 698.885,A -85,B 0,C 180,E1 540.352,E2 540.352} C_VEL
LIN {X 0,Y 607.953,Z 686.452,A -85,B 0,C 180,E1 542.664,E2 542.664} C_VEL
LIN {X 0,Y 607.994,Z 669.89,A -85,B 0,C 180,E1 544.623,E2 544.623} C_VEL
LIN {X 0,Y 608.06,Z 648.143,A -85,B 0,C 180,E1 546.32,E2 546.32} C_VEL
LIN {X 0,Y 608.111,Z 623.286,A -85,B 0,C 180,E1 547.527,E2 547.527} C_VEL
LIN {X 0,Y 608.168,Z 596.73,A -85,B 0,C 180,E1 548.199,E2 548.199} C_VEL
LIN {X 0,Y 607.784,Z 549.53,A -85,B 0,C 180,E1 548.837,E2 548.837} C_VEL
LIN {X 0,Y 607.611,Z 549.53,A -85,B 0,C 180,E1 554.377,E2 554.377} C_VEL
LIN {X 0,Y 607.787,Z 549.53,A -85,B 0,C 180,E1 560.337,E2 560.337} C_VEL
LIN {X 0,Y 607.759,Z 549.53,A -85,B 0,C 180,E1 564.964,E2 564.964} C_VEL
LIN {X 0,Y 607.597,Z 549.53,A -85,B 0,C 180,E1 569.78,E2 569.78} C_VEL
LIN {X 0,Y 607.609,Z 549.53,A -85,B 0,C 180,E1 576.584,E2 576.584} C_VEL
LIN {X 0,Y 607.613,Z 549.53,A -85,B 0,C 180,E1 582.105,E2 582.105} C_VEL
LIN {X 0,Y 607.277,Z 549.53,A -85,B 0,C 180,E1 587.856,E2 587.856} C_VEL
LIN {X 0,Y 607.286,Z 549.53,A -85,B 0,C 180,E1 592.665,E2 592.665} C_VEL
LIN {X 0,Y 607.68,Z 549.53,A -85,B 0,C 180,E1 597.592,E2 597.592} C_VEL
LIN {X 0,Y 607.91,Z 550.319,A -85,B 0,C 180,E1 600.425,E2 600.425} C_VEL
LIN {X 0,Y 608.59,Z 622.463,A -85,B 0,C 180,E1 601.537,E2 601.537} C_VEL
LIN {X 0,Y 608.562,Z 661.79,A -85,B 0,C 180,E1 602.73,E2 602.73} C_VEL
LIN {X 0,Y 608.418,Z 699.372,A -85,B 0,C 180,E1 604.47,E2 604.47} C_VEL
LIN {X 0,Y 608.267,Z 735.646,A -85,B 0,C 180,E1 606.804,E2 606.804} C_VEL
LIN {X 0,Y 608.118,Z 767.02,A -85,B 0,C 180,E1 609.479,E2 609.479} C_VEL
LIN {X 0,Y 608.023,Z 794.219,A -85,B 0,C 180,E1 612.485,E2 612.485} C_VEL
LIN {X 0,Y 607.886,Z 817.245,A -85,B 0,C 180,E1 615.808,E2 615.808} C_VEL
LIN {X 0,Y 607.819,Z 834.972,A -85,B 0,C 180,E1 619.267,E2 619.267} C_VEL
LIN {X 0,Y 607.79,Z 847.676,A -85,B 0,C 180,E1 622.868,E2 622.868} C_VEL
LIN {X 0,Y 607.671,Z 853.955,A -85,B 0,C 180,E1 625.727,E2 625.727} C_VEL
LIN {X 0,Y 607.712,Z 857.086,A -85,B 0,C 180,E1 628.577,E2 628.577} C_VEL
LIN {X 0,Y 607.889,Z 857.086,A -85,B 0,C 180,E1 631.422,E2 631.422} C_VEL
LIN {X 0,Y 607.927,Z 852.756,A -85,B 0,C 180,E1 634.984,E2 634.984} C_VEL
LIN {X 0,Y 607.878,Z 842.07,A -85,B 0,C 180,E1 638.926,E2 638.926} C_VEL
LIN {X 0,Y 607.905,Z 826.445,A -85,B 0,C 180,E1 642.546,E2 642.546} C_VEL
LIN {X 0,Y 607.957,Z 805.339,A -85,B 0,C 180,E1 646.031,E2 646.031} C_VEL
LIN {X 0,Y 608.034,Z 779.192,A -85,B 0,C 180,E1 649.271,E2 649.271} C_VEL
LIN {X 0,Y 608.171,Z 749,A -85,B 0,C 180,E1 652.14,E2 652.14} C_VEL
LIN {X 0,Y 608.308,Z 715.852,A -85,B 0,C 180,E1 654.554,E2 654.554} C_VEL
LIN {X 0,Y 608.483,Z 679.683,A -85,B 0,C 180,E1 656.515,E2 656.515} C_VEL
LIN {X 0,Y 608.573,Z 642.885,A -85,B 0,C 180,E1 657.914,E2 657.914} C_VEL
LIN {X 0,Y 608.663,Z 606.946,A -85,B 0,C 180,E1 658.762,E2 658.762} C_VEL
LIN {X 0,Y 607.897,Z 549.53,A -85,B 0,C 180,E1 659.625,E2 659.625} C_VEL
LIN {X 0,Y 607.676,Z 549.53,A -85,B 0,C 180,E1 666.587,E2 666.587} C_VEL
LIN {X 0,Y 607.349,Z 549.53,A -85,B 0,C 180,E1 671.813,E2 671.813} C_VEL
LIN {X 0,Y 607.514,Z 549.53,A -85,B 0,C 180,E1 676.088,E2 676.088} C_VEL
LIN {X 0,Y 607.451,Z 549.53,A -85,B 0,C 180,E1 680.369,E2 680.369} C_VEL
LIN {X 0,Y 607.427,Z 549.53,A -85,B 0,C 180,E1 685.157,E2 685.157} C_VEL
LIN {X 0,Y 607.575,Z 549.53,A -85,B 0,C 180,E1 690.386,E2 690.386} C_VEL
LIN {X 0,Y 607.798,Z 549.53,A -85,B 0,C 180,E1 695.038,E2 695.038} C_VEL
LIN {X 0,Y 607.719,Z 549.717,A -85,B 0,C 180,E1 699.988,E2 699.988} C_VEL
LIN {X 0,Y 608.164,Z 591.253,A -85,B 0,C 180,E1 700.631,E2 700.631} C_VEL
LIN {X 0,Y 608.13,Z 619.797,A -85,B 0,C 180,E1 701.653,E2 701.653} C_VEL
LIN {X 0,Y 608.041,Z 646.415,A -85,B 0,C 180,E1 703.235,E2 703.235} C_VEL
LIN {X 0,Y 608.005,Z 667.454,A -85,B 0,C 180,E1 705.092,E2 705.092} C_VEL
LIN {X 0,Y 607.94,Z 685.731,A -85,B 0,C 180,E1 707.459,E2 707.459} C_VEL
LIN {X 0,Y 607.894,Z 698.322,A -85,B 0,C 180,E1 709.996,E2 709.996} C_VEL
LIN {X 0,Y 607.946,Z 704.615,A -85,B 0,C 180,E1 712.157,E2 712.157} C_VEL
LIN {X 0,Y 607.918,Z 707.345,A -85,B 0,C 180,E1 714.305,E2 714.305} C_VEL
LIN {X 0,Y 607.942,Z 705.702,A -85,B 0,C 180,E1 717.158,E2 717.158} C_VEL
LIN {X 0,Y 607.926,Z 697.986,A -85,B 0,C 180,E1 720.003,E2 720.003} C_VEL
LIN {X 0,Y 608.012,Z 684.333,A -85,B 0,C 180,E1 722.671,E2 722.671} C_VEL
LIN {X 0,Y 607.998,Z 665.818,A -85,B 0,C 180,E1 724.987,E2 724.987} C_VEL
LIN {X 0,Y 608.079,Z 643.249,A -85,B 0,C 180,E1 726.904,E2 726.904} C_VEL
LIN {X 0,Y 608.095,Z 616.982,A -85,B 0,C 180,E1 728.386,E2 728.386} C_VEL
LIN {X 0,Y 608.175,Z 589.035,A -85,B 0,C 180,E1 729.33,E2 729.33} C_VEL
LIN {X 0,Y 607.461,Z 549.53,A -85,B 0,C 180,E1 729.972,E2 729.972} C_VEL
LIN {X 0,Y 607.895,Z 549.53,A -85,B 0,C 180,E1 732.913,E2 732.913} C_VEL
LIN {X 0,Y 607.612,Z 549.53,A -85,B 0,C 180,E1 738.839,E2 738.839} C_VEL
LIN {X 0,Y 607.574,Z 549.53,A -85,B 0,C 180,E1 743.419,E2 743.419} C_VEL
LIN {X 0,Y 607.68,Z 549.53,A -85,B 0,C 180,E1 748.156,E2 748.156} C_VEL
LIN {X 0,Y 607.808,Z 549.53,A -85,B 0,C 180,E1 753.111,E2 753.111} C_VEL
LIN {X 0,Y 607.484,Z 549.53,A -85,B 0,C 180,E1 759.634,E2 759.634} C_VEL
LIN {X 0,Y 607.544,Z 549.53,A -85,B 0,C 180,E1 765.93,E2 765.93} C_VEL
LIN {X 0,Y 607.417,Z 549.53,A -85,B 0,C 180,E1 770.372,E2 770.372} C_VEL
LIN {X 0,Y 607.403,Z 549.53,A -85,B 0,C 180,E1 775.148,E2 775.148} C_VEL
LIN {X 0,Y 607.528,Z 549.53,A -85,B 0,C 180,E1 780.391,E2 780.391} C_VEL
LIN {X 0,Y 607.874,Z 549.53,A -85,B 0,C 180,E1 785.035,E2 785.035} C_VEL
LIN {X 0,Y 607.802,Z 549.53,A -85,B 0,C 180,E1 787.942,E2 787.942} C_VEL
LIN {X 0,Y 608.405,Z 590.825,A -85,B 0,C 180,E1 788.872,E2 788.872} C_VEL
LIN {X 0,Y 608.333,Z 626.091,A -85,B 0,C 180,E1 790.208,E2 790.208} C_VEL
LIN {X 0,Y 608.232,Z 660.471,A -85,B 0,C 180,E1 792.118,E2 792.118} C_VEL
LIN {X 0,Y 608.085,Z 691.753,A -85,B 0,C 180,E1 794.527,E2 794.527} C_VEL
LIN {X 0,Y 607.968,Z 718.509,A -85,B 0,C 180,E1 797.273,E2 797.273} C_VEL
LIN {X 0,Y 607.886,Z 740.849,A -85,B 0,C 180,E1 800.353,E2 800.353} C_VEL
LIN {X 0,Y 607.842,Z 757.745,A -85,B 0,C 180,E1 803.585,E2 803.585} C_VEL
LIN {X 0,Y 607.958,Z 768.13,A -85,B 0,C 180,E1 806.442,E2 806.442} C_VEL
LIN {X 0,Y 607.863,Z 775.549,A -85,B 0,C 180,E1 810,E2 810} C_VEL
LIN {X 0,Y 607.82,Z 777.483,A -85,B 0,C 180,E1 812.847,E2 812.847} C_VEL
LIN {X 0,Y 607.782,Z 775.798,A -85,B 0,C 180,E1 815.7,E2 815.7} C_VEL
LIN {X 0,Y 607.832,Z 768.619,A -85,B 0,C 180,E1 819.288,E2 819.288} C_VEL
LIN {X 0,Y 607.836,Z 756.801,A -85,B 0,C 180,E1 822.548,E2 822.548} C_VEL
LIN {X 0,Y 607.914,Z 739.028,A -85,B 0,C 180,E1 825.848,E2 825.848} C_VEL
LIN {X 0,Y 607.975,Z 715.675,A -85,B 0,C 180,E1 828.963,E2 828.963} C_VEL
LIN {X 0,Y 608.115,Z 687.488,A -85,B 0,C 180,E1 831.76,E2 831.76} C_VEL
LIN {X 0,Y 608.222,Z 656.047,A -85,B 0,C 180,E1 834.071,E2 834.071} C_VEL
LIN {X 0,Y 608.3,Z 621.121,A -85,B 0,C 180,E1 835.93,E2 835.93} C_VEL
LIN {X 0,Y 608.362,Z 584.071,A -85,B 0,C 180,E1 837.235,E2 837.235} C_VEL
LIN {X 0,Y 607.59,Z 552.59,A -85,B 0,C 180,E1 837.903,E2 837.903} C_VEL
LIN {X 0,Y 607.316,Z 549.53,A -85,B 0,C 180,E1 837.976,E2 837.976} C_VEL
LIN {X 0,Y 607.945,Z 549.53,A -85,B 0,C 180,E1 843.103,E2 843.103} C_VEL
LIN {X 0,Y 607.561,Z 549.53,A -85,B 0,C 180,E1 848.389,E2 848.389} C_VEL
LIN {X 0,Y 607.688,Z 549.53,A -85,B 0,C 180,E1 852.109,E2 852.109} C_VEL
LIN {X 0,Y 607.773,Z 549.53,A -85,B 0,C 180,E1 858.154,E2 858.154} C_VEL
LIN {X 0,Y 607.617,Z 549.53,A -85,B 0,C 180,E1 863.409,E2 863.409} C_VEL
LIN {X 0,Y 607.599,Z 549.53,A -85,B 0,C 180,E1 867.62,E2 867.62} C_VEL
LIN {X 0,Y 607.564,Z 549.53,A -85,B 0,C 180,E1 871.838,E2 871.838} C_VEL
LIN {X 0,Y 607.546,Z 549.53,A -85,B 0,C 180,E1 878.122,E2 878.122} C_VEL
LIN {X 0,Y 607.859,Z 549.53,A -85,B 0,C 180,E1 882.665,E2 882.665} C_VEL
LIN {X 0,Y 606.263,Z 549.53,A -85,B 0,C 180,E1 883.084,E2 883.084} C_VEL
LIN {X 0,Y 608.105,Z 574.972,A -85,B 0,C 180,E1 883.444,E2 883.444} C_VEL
LIN {X 0,Y 608.112,Z 611.663,A -85,B 0,C 180,E1 884.017,E2 884.017} C_VEL
LIN {X 0,Y 608.074,Z 636.7,A -85,B 0,C 180,E1 884.956,E2 884.956} C_VEL
LIN {X 0,Y 608.014,Z 660.322,A -85,B 0,C 180,E1 886.45,E2 886.45} C_VEL
LIN {X 0,Y 607.937,Z 679.812,A -85,B 0,C 180,E1 888.361,E2 888.361} C_VEL
LIN {X 0,Y 607.894,Z 693.185,A -85,B 0,C 180,E1 890.351,E2 890.351} C_VEL
LIN {X 0,Y 607.884,Z 703.3,A -85,B 0,C 180,E1 892.867,E2 892.867} C_VEL
LIN {X 0,Y 607.976,Z 706.308,A -85,B 0,C 180,E1 894.299,E2 894.299} C_VEL
LIN {X 0,Y 607.848,Z 707.453,A -85,B 0,C 180,E1 895.728,E2 895.728} C_VEL
LIN {X 0,Y 605.265,Z 707.068,A -85,B 0,C 180,E1 896.946,E2 896.946} C_VEL
LIN {X 0,Y 600.075,Z 704.177,A -85,B 0,C 180,E1 898.748,E2 898.748} C_VEL
LIN {X 0,Y 600.017,Z 703.596,A -85,B 0,C 180,E1 898.953,E2 898.953} C_VEL
LIN {X 0,Y 600.054,Z 694.215,A -85,B 0,C 180,E1 901.438,E2 901.438} C_VEL
LIN {X 0,Y 600.126,Z 678.74,A -85,B 0,C 180,E1 903.781,E2 903.781} C_VEL
LIN {X 0,Y 600.234,Z 658.016,A -85,B 0,C 180,E1 905.768,E2 905.768} C_VEL
LIN {X 0,Y 600.333,Z 634.259,A -85,B 0,C 180,E1 907.217,E2 907.217} C_VEL
LIN {X 0,Y 600.412,Z 608.742,A -85,B 0,C 180,E1 908.124,E2 908.124} C_VEL
LIN {X 0,Y 599.95,Z 549.53,A -85,B 0,C 180,E1 908.95,E2 908.95} C_VEL
LIN {X 0,Y 599.695,Z 549.53,A -85,B 0,C 180,E1 914.571,E2 914.571} C_VEL
LIN {X 0,Y 599.766,Z 549.53,A -85,B 0,C 180,E1 920.621,E2 920.621} C_VEL
LIN {X 0,Y 599.729,Z 549.53,A -85,B 0,C 180,E1 925.321,E2 925.321} C_VEL
LIN {X 0,Y 599.524,Z 549.53,A -85,B 0,C 180,E1 931.142,E2 931.142} C_VEL
LIN {X 0,Y 599.644,Z 549.53,A -85,B 0,C 180,E1 937.151,E2 937.151} C_VEL
LIN {X 0,Y 599.583,Z 549.53,A -85,B 0,C 180,E1 943.118,E2 943.118} C_VEL
LIN {X 0,Y 599.42,Z 549.53,A -85,B 0,C 180,E1 949.11,E2 949.11} C_VEL
LIN {X 0,Y 599.3,Z 549.53,A -85,B 0,C 180,E1 953.678,E2 953.678} C_VEL
LIN {X 0,Y 599.726,Z 549.53,A -85,B 0,C 180,E1 958.099,E2 958.099} C_VEL
LIN {X 0,Y 599.854,Z 549.53,A -85,B 0,C 180,E1 959.974,E2 959.974} C_VEL
LIN {X 0,Y 601.388,Z 557.163,A -85,B 0,C 180,E1 960.164,E2 960.164} C_VEL
LIN {X 0,Y 601.625,Z 623.421,A -85,B 0,C 180,E1 961.199,E2 961.199} C_VEL
LIN {X 0,Y 601.446,Z 662.577,A -85,B 0,C 180,E1 962.41,E2 962.41} C_VEL
LIN {X 0,Y 601.134,Z 701.156,A -85,B 0,C 180,E1 964.238,E2 964.238} C_VEL
LIN {X 0,Y 600.77,Z 736.702,A -85,B 0,C 180,E1 966.58,E2 966.58} C_VEL
LIN {X 0,Y 600.477,Z 768.934,A -85,B 0,C 180,E1 969.398,E2 969.398} C_VEL
LIN {X 0,Y 600.274,Z 795.689,A -85,B 0,C 180,E1 972.44,E2 972.44} C_VEL
LIN {X 0,Y 600.064,Z 818.35,A -85,B 0,C 180,E1 975.807,E2 975.807} C_VEL
LIN {X 0,Y 599.962,Z 835.867,A -85,B 0,C 180,E1 979.338,E2 979.338} C_VEL
LIN {X 0,Y 599.89,Z 847.679,A -85,B 0,C 180,E1 982.773,E2 982.773} C_VEL
LIN {X 0,Y 599.784,Z 853.958,A -85,B 0,C 180,E1 985.671,E2 985.671} C_VEL
LIN {X 0,Y 599.811,Z 857.088,A -85,B 0,C 180,E1 988.558,E2 988.558} C_VEL
LIN {X 0,Y 599.983,Z 857.088,A -85,B 0,C 180,E1 991.441,E2 991.441} C_VEL
LIN {X 0,Y 600.013,Z 852.756,A -85,B 0,C 180,E1 995.05,E2 995.05} C_VEL
LIN {X 0,Y 599.977,Z 842.073,A -85,B 0,C 180,E1 999.045,E2 999.045} C_VEL
LIN {X 0,Y 600.04,Z 826.448,A -85,B 0,C 180,E1 1002.713,E2 1002.713} C_VEL
LIN {X 0,Y 600.117,Z 804.707,A -85,B 0,C 180,E1 1006.336,E2 1006.336} C_VEL
LIN {X 0,Y 600.367,Z 779.029,A -85,B 0,C 180,E1 1009.546,E2 1009.546} C_VEL
LIN {X 0,Y 600.65,Z 748.436,A -85,B 0,C 180,E1 1012.481,E2 1012.481} C_VEL
LIN {X 0,Y 600.984,Z 713.878,A -85,B 0,C 180,E1 1015.003,E2 1015.003} C_VEL
LIN {X 0,Y 601.37,Z 675.782,A -85,B 0,C 180,E1 1017.039,E2 1017.039} C_VEL
LIN {X 0,Y 601.585,Z 636.407,A -85,B 0,C 180,E1 1018.466,E2 1018.466} C_VEL
LIN {X 0,Y 601.746,Z 597.173,A -85,B 0,C 180,E1 1019.278,E2 1019.278} C_VEL
LIN {X 0,Y 600.781,Z 553.099,A -85,B 0,C 180,E1 1019.924,E2 1019.924} C_VEL
LIN {X 0,Y 599.896,Z 549.53,A -85,B 0,C 180,E1 1020.026,E2 1020.026} C_VEL
LIN {X 0,Y 599.743,Z 549.53,A -85,B 0,C 180,E1 1027.152,E2 1027.152} C_VEL
LIN {X 0,Y 599.427,Z 549.53,A -85,B 0,C 180,E1 1033.113,E2 1033.113} C_VEL
LIN {X 0,Y 599.601,Z 549.53,A -85,B 0,C 180,E1 1039.033,E2 1039.033} C_VEL
LIN {X 0,Y 599.572,Z 549.53,A -85,B 0,C 180,E1 1044.633,E2 1044.633} C_VEL
LIN {X 0,Y 599.631,Z 549.53,A -85,B 0,C 180,E1 1049.784,E2 1049.784} C_VEL
LIN {X 0,Y 599.877,Z 549.53,A -85,B 0,C 180,E1 1054.916,E2 1054.916} C_VEL
LIN {X 0,Y 599.92,Z 549.53,A -85,B 0,C 180,E1 1059.78,E2 1059.78} C_VEL
LIN {X 0,Y 600.493,Z 590.445,A -85,B 0,C 180,E1 1060.424,E2 1060.424} C_VEL
LIN {X 0,Y 600.418,Z 618.337,A -85,B 0,C 180,E1 1061.409,E2 1061.409} C_VEL
LIN {X 0,Y 600.268,Z 644.525,A -85,B 0,C 180,E1 1062.942,E2 1062.942} C_VEL
LIN {X 0,Y 600.174,Z 666.691,A -85,B 0,C 180,E1 1064.882,E2 1064.882} C_VEL
LIN {X 0,Y 600.081,Z 685.312,A -85,B 0,C 180,E1 1067.292,E2 1067.292} C_VEL
LIN {X 0,Y 600,Z 698.077,A -85,B 0,C 180,E1 1069.863,E2 1069.863} C_VEL
LIN {X 0,Y 600.048,Z 704.474,A -85,B 0,C 180,E1 1072.053,E2 1072.053} C_VEL
LIN {X 0,Y 600.038,Z 707.3,A -85,B 0,C 180,E1 1074.23,E2 1074.23} C_VEL
LIN {X 0,Y 600.044,Z 705.808,A -85,B 0,C 180,E1 1077.12,E2 1077.12} C_VEL
LIN {X 0,Y 600.03,Z 698.232,A -85,B 0,C 180,E1 1080.003,E2 1080.003} C_VEL
LIN {X 0,Y 600.105,Z 685.879,A -85,B 0,C 180,E1 1082.525,E2 1082.525} C_VEL
LIN {X 0,Y 600.171,Z 668.169,A -85,B 0,C 180,E1 1084.871,E2 1084.871} C_VEL
LIN {X 0,Y 600.263,Z 645.284,A -85,B 0,C 180,E1 1086.914,E2 1086.914} C_VEL
LIN {X 0,Y 600.363,Z 618.492,A -85,B 0,C 180,E1 1088.495,E2 1088.495} C_VEL
LIN {X 0,Y 600.526,Z 589.916,A -85,B 0,C 180,E1 1089.495,E2 1089.495} C_VEL
LIN {X 0,Y 599.728,Z 549.53,A -85,B 0,C 180,E1 1090.148,E2 1090.148} C_VEL
LIN {X 0,Y 599.534,Z 549.53,A -85,B 0,C 180,E1 1094.582,E2 1094.582} C_VEL
LIN {X 0,Y 599.677,Z 549.53,A -85,B 0,C 180,E1 1099.098,E2 1099.098} C_VEL
LIN {X 0,Y 599.589,Z 549.53,A -85,B 0,C 180,E1 1103.75,E2 1103.75} C_VEL
LIN {X 0,Y 599.652,Z 549.53,A -85,B 0,C 180,E1 1108.568,E2 1108.568} C_VEL
LIN {X 0,Y 599.683,Z 549.53,A -85,B 0,C 180,E1 1113.852,E2 1113.852} C_VEL
LIN {X 0,Y 599.589,Z 549.53,A -85,B 0,C 180,E1 1118.995,E2 1118.995} C_VEL
LIN {X 0,Y 599.55,Z 549.53,A -85,B 0,C 180,E1 1125.186,E2 1125.186} C_VEL
LIN {X 0,Y 599.523,Z 549.53,A -85,B 0,C 180,E1 1131,E2 1131} C_VEL
LIN {X 0,Y 599.54,Z 549.53,A -85,B 0,C 180,E1 1134.623,E2 1134.623} C_VEL
LIN {X 0,Y 599.59,Z 549.53,A -85,B 0,C 180,E1 1139.775,E2 1139.775} C_VEL
LIN {X 0,Y 599.938,Z 549.53,A -85,B 0,C 180,E1 1144.9,E2 1144.9} C_VEL
LIN {X 0,Y 599.95,Z 549.53,A -85,B 0,C 180,E1 1147.613,E2 1147.613} C_VEL
LIN {X 0,Y 601.345,Z 566.62,A -85,B 0,C 180,E1 1147.967,E2 1147.967} C_VEL
LIN {X 0,Y 601.131,Z 603,A -85,B 0,C 180,E1 1148.965,E2 1148.965} C_VEL
LIN {X 0,Y 600.89,Z 638.729,A -85,B 0,C 180,E1 1150.545,E2 1150.545} C_VEL
LIN {X 0,Y 600.576,Z 672.786,A -85,B 0,C 180,E1 1152.719,E2 1152.719} C_VEL
LIN {X 0,Y 600.317,Z 702.169,A -85,B 0,C 180,E1 1155.273,E2 1155.273} C_VEL
LIN {X 0,Y 600.098,Z 727.52,A -85,B 0,C 180,E1 1158.21,E2 1158.21} C_VEL
LIN {X 0,Y 599.949,Z 747.378,A -85,B 0,C 180,E1 1161.319,E2 1161.319} C_VEL
LIN {X 0,Y 599.867,Z 762.253,A -85,B 0,C 180,E1 1164.587,E2 1164.587} C_VEL
LIN {X 0,Y 599.872,Z 771.847,A -85,B 0,C 180,E1 1167.838,E2 1167.838} C_VEL
LIN {X 0,Y 599.829,Z 776.965,A -85,B 0,C 180,E1 1171.442,E2 1171.442} C_VEL
LIN {X 0,Y 599.924,Z 777.059,A -85,B 0,C 180,E1 1174.328,E2 1174.328} C_VEL
LIN {X 0,Y 599.89,Z 772.101,A -85,B 0,C 180,E1 1177.954,E2 1177.954} C_VEL
LIN {X 0,Y 599.909,Z 762.835,A -85,B 0,C 180,E1 1181.165,E2 1181.165} C_VEL
LIN {X 0,Y 599.971,Z 747.481,A -85,B 0,C 180,E1 1184.569,E2 1184.569} C_VEL
LIN {X 0,Y 600.081,Z 727.142,A -85,B 0,C 180,E1 1187.755,E2 1187.755} C_VEL
LIN {X 0,Y 600.355,Z 701.272,A -85,B 0,C 180,E1 1190.726,E2 1190.726} C_VEL
LIN {X 0,Y 600.617,Z 670.888,A -85,B 0,C 180,E1 1193.334,E2 1193.334} C_VEL
LIN {X 0,Y 600.892,Z 636.984,A -85,B 0,C 180,E1 1195.454,E2 1195.454} C_VEL
LIN {X 0,Y 601.151,Z 603.37,A -85,B 0,C 180,E1 1196.932,E2 1196.932} C_VEL
LIN {X 0,Y 601.318,Z 569.16,A -85,B 0,C 180,E1 1197.892,E2 1197.892} C_VEL
LIN {X 0,Y 600.104,Z 552.735,A -85,B 0,C 180,E1 1198.233,E2 1198.233} C_VEL
LIN {X 0,Y 599.422,Z 549.53,A -85,B 0,C 180,E1 1198.369,E2 1198.369} C_VEL
LIN {X 0,Y 599.831,Z 549.53,A -85,B 0,C 180,E1 1203.875,E2 1203.875} C_VEL
LIN {X 0,Y 599.54,Z 549.53,A -85,B 0,C 180,E1 1208.999,E2 1208.999} C_VEL
LIN {X 0,Y 599.479,Z 549.53,A -85,B 0,C 180,E1 1213.109,E2 1213.109} C_VEL
LIN {X 0,Y 599.584,Z 549.53,A -85,B 0,C 180,E1 1219.124,E2 1219.124} C_VEL
LIN {X 0,Y 599.722,Z 549.53,A -85,B 0,C 180,E1 1224.635,E2 1224.635} C_VEL
LIN {X 0,Y 599.595,Z 549.53,A -85,B 0,C 180,E1 1229.774,E2 1229.774} C_VEL
LIN {X 0,Y 599.364,Z 549.53,A -85,B 0,C 180,E1 1235.022,E2 1235.022} C_VEL
LIN {X 0,Y 599.34,Z 549.53,A -85,B 0,C 180,E1 1239.357,E2 1239.357} C_VEL
LIN {X 0,Y 599.205,Z 549.53,A -85,B 0,C 180,E1 1242.721,E2 1242.721} C_VEL
LIN {X 0,Y 598.553,Z 549.53,A -85,B 0,C 180,E1 1242.921,E2 1242.921} C_VEL
LIN {X 0,Y 600.404,Z 574.54,A -85,B 0,C 180,E1 1243.276,E2 1243.276} C_VEL
LIN {X 0,Y 600.4,Z 611.02,A -85,B 0,C 180,E1 1243.844,E2 1243.844} C_VEL
LIN {X 0,Y 600.292,Z 636.168,A -85,B 0,C 180,E1 1244.785,E2 1244.785} C_VEL
LIN {X 0,Y 600.186,Z 659.629,A -85,B 0,C 180,E1 1246.27,E2 1246.27} C_VEL
LIN {X 0,Y 600.09,Z 679.378,A -85,B 0,C 180,E1 1248.207,E2 1248.207} C_VEL
LIN {X 0,Y 600.023,Z 692.894,A -85,B 0,C 180,E1 1250.223,E2 1250.223} C_VEL
LIN {X 0,Y 599.99,Z 703.161,A -85,B 0,C 180,E1 1252.772,E2 1252.772} C_VEL
LIN {X 0,Y 600.094,Z 706.225,A -85,B 0,C 180,E1 1254.224,E2 1254.224} C_VEL
LIN {X 0,Y 599.954,Z 707.423,A -85,B 0,C 180,E1 1255.722,E2 1255.722} C_VEL
LIN {X 0,Y 599.985,Z 705.985,A -85,B 0,C 180,E1 1257.835,E2 1257.835} C_VEL
LIN {X 0,Y 600.017,Z 703.596,A -85,B 0,C 180,E1 1258.953,E2 1258.953} C_VEL
LIN {X 0,Y 597.687,Z 700.057,A -85,B 0,C 180,E1 1260.142,E2 1260.142} C_VEL
LIN {X 0,Y 592.375,Z 692.544,A -85,B 0,C 180,E1 1261.839,E2 1261.839} C_VEL
LIN {X 0,Y 592.244,Z 691.482,A -85,B 0,C 180,E1 1262.025,E2 1262.025} C_VEL
LIN {X 0,Y 592.281,Z 676.046,A -85,B 0,C 180,E1 1264.197,E2 1264.197} C_VEL
LIN {X 0,Y 592.431,Z 656.109,A -85,B 0,C 180,E1 1266.042,E2 1266.042} C_VEL
LIN {X 0,Y 592.569,Z 631.517,A -85,B 0,C 180,E1 1267.496,E2 1267.496} C_VEL
LIN {X 0,Y 592.694,Z 605.167,A -85,B 0,C 180,E1 1268.369,E2 1268.369} C_VEL
LIN {X 0,Y 592.102,Z 549.53,A -85,B 0,C 180,E1 1269.128,E2 1269.128} C_VEL
LIN {X 0,Y 591.788,Z 549.53,A -85,B 0,C 180,E1 1274.77,E2 1274.77} C_VEL
LIN {X 0,Y 591.79,Z 549.53,A -85,B 0,C 180,E1 1280.912,E2 1280.912} C_VEL
LIN {X 0,Y 591.518,Z 549.53,A -85,B 0,C 180,E1 1286.75,E2 1286.75} C_VEL
LIN {X 0,Y 591.646,Z 549.53,A -85,B 0,C 180,E1 1290.667,E2 1290.667} C_VEL
LIN {X 0,Y 591.689,Z 549.53,A -85,B 0,C 180,E1 1295.911,E2 1295.911} C_VEL
LIN {X 0,Y 591.655,Z 549.53,A -85,B 0,C 180,E1 1301.535,E2 1301.535} C_VEL
LIN {X 0,Y 591.51,Z 549.53,A -85,B 0,C 180,E1 1306.458,E2 1306.458} C_VEL
LIN {X 0,Y 591.519,Z 549.53,A -85,B 0,C 180,E1 1312.259,E2 1312.259} C_VEL
LIN {X 0,Y 591.783,Z 549.53,A -85,B 0,C 180,E1 1317.619,E2 1317.619} C_VEL
LIN {X 0,Y 591.868,Z 549.53,A -85,B 0,C 180,E1 1319.528,E2 1319.528} C_VEL
LIN {X 0,Y 594.573,Z 559.952,A -85,B 0,C 180,E1 1319.825,E2 1319.825} C_VEL
LIN {X 0,Y 594.679,Z 623.747,A -85,B 0,C 180,E1 1320.838,E2 1320.838} C_VEL
LIN {X 0,Y 594.368,Z 663.386,A -85,B 0,C 180,E1 1322.086,E2 1322.086} C_VEL
LIN {X 0,Y 593.888,Z 701.137,A -85,B 0,C 180,E1 1323.899,E2 1323.899} C_VEL
LIN {X 0,Y 593.308,Z 736.957,A -85,B 0,C 180,E1 1326.287,E2 1326.287} C_VEL
LIN {X 0,Y 592.861,Z 768.938,A -85,B 0,C 180,E1 1329.122,E2 1329.122} C_VEL
LIN {X 0,Y 592.533,Z 795.693,A -85,B 0,C 180,E1 1332.203,E2 1332.203} C_VEL
LIN {X 0,Y 592.204,Z 817.816,A -85,B 0,C 180,E1 1335.521,E2 1335.521} C_VEL
LIN {X 0,Y 592.025,Z 834.248,A -85,B 0,C 180,E1 1338.801,E2 1338.801} C_VEL
LIN {X 0,Y 591.971,Z 846.713,A -85,B 0,C 180,E1 1342.308,E2 1342.308} C_VEL
LIN {X 0,Y 591.883,Z 853.961,A -85,B 0,C 180,E1 1345.613,E2 1345.613} C_VEL
LIN {X 0,Y 591.91,Z 857.09,A -85,B 0,C 180,E1 1348.539,E2 1348.539} C_VEL
LIN {X 0,Y 592.077,Z 857.09,A -85,B 0,C 180,E1 1351.46,E2 1351.46} C_VEL
LIN {X 0,Y 592.111,Z 852.755,A -85,B 0,C 180,E1 1355.118,E2 1355.118} C_VEL
LIN {X 0,Y 592.092,Z 842.076,A -85,B 0,C 180,E1 1359.166,E2 1359.166} C_VEL
LIN {X 0,Y 592.188,Z 826.451,A -85,B 0,C 180,E1 1362.885,E2 1362.885} C_VEL
LIN {X 0,Y 592.352,Z 804.941,A -85,B 0,C 180,E1 1366.523,E2 1366.523} C_VEL
LIN {X 0,Y 592.714,Z 778.959,A -85,B 0,C 180,E1 1369.817,E2 1369.817} C_VEL
LIN {X 0,Y 593.143,Z 748.739,A -85,B 0,C 180,E1 1372.756,E2 1372.756} C_VEL
LIN {X 0,Y 593.645,Z 714.669,A -85,B 0,C 180,E1 1375.282,E2 1375.282} C_VEL
LIN {X 0,Y 594.218,Z 676.9,A -85,B 0,C 180,E1 1377.339,E2 1377.339} C_VEL
LIN {X 0,Y 594.612,Z 637.614,A -85,B 0,C 180,E1 1378.797,E2 1378.797} C_VEL
LIN {X 0,Y 594.857,Z 598.957,A -85,B 0,C 180,E1 1379.624,E2 1379.624} C_VEL
LIN {X 0,Y 594.013,Z 555.438,A -85,B 0,C 180,E1 1380.268,E2 1380.268} C_VEL
LIN {X 0,Y 591.868,Z 549.53,A -85,B 0,C 180,E1 1380.475,E2 1380.475} C_VEL
LIN {X 0,Y 591.74,Z 549.53,A -85,B 0,C 180,E1 1385.915,E2 1385.915} C_VEL
LIN {X 0,Y 591.599,Z 549.53,A -85,B 0,C 180,E1 1390.078,E2 1390.078} C_VEL
LIN {X 0,Y 591.609,Z 549.53,A -85,B 0,C 180,E1 1395.583,E2 1395.583} C_VEL
LIN {X 0,Y 591.594,Z 549.53,A -85,B 0,C 180,E1 1400.384,E2 1400.384} C_VEL
LIN {X 0,Y 591.657,Z 549.53,A -85,B 0,C 180,E1 1404.71,E2 1404.71} C_VEL
LIN {X 0,Y 591.578,Z 549.53,A -85,B 0,C 180,E1 1411.014,E2 1411.014} C_VEL
LIN {X 0,Y 591.686,Z 549.53,A -85,B 0,C 180,E1 1415.92,E2 1415.92} C_VEL
LIN {X 0,Y 592.002,Z 549.53,A -85,B 0,C 180,E1 1419.577,E2 1419.577} C_VEL
LIN {X 0,Y 592.844,Z 591.5,A -85,B 0,C 180,E1 1420.26,E2 1420.26} C_VEL
LIN {X 0,Y 592.697,Z 618.869,A -85,B 0,C 180,E1 1421.254,E2 1421.254} C_VEL
LIN {X 0,Y 592.495,Z 645.286,A -85,B 0,C 180,E1 1422.839,E2 1422.839} C_VEL
LIN {X 0,Y 592.333,Z 667.814,A -85,B 0,C 180,E1 1424.866,E2 1424.866} C_VEL
LIN {X 0,Y 592.199,Z 686.019,A -85,B 0,C 180,E1 1427.307,E2 1427.307} C_VEL
LIN {X 0,Y 592.121,Z 697.833,A -85,B 0,C 180,E1 1429.727,E2 1429.727} C_VEL
LIN {X 0,Y 592.159,Z 704.334,A -85,B 0,C 180,E1 1431.946,E2 1431.946} C_VEL
LIN {X 0,Y 592.127,Z 707.249,A -85,B 0,C 180,E1 1434.152,E2 1434.152} C_VEL
LIN {X 0,Y 592.138,Z 705.914,A -85,B 0,C 180,E1 1437.082,E2 1437.082} C_VEL
LIN {X 0,Y 592.134,Z 698.477,A -85,B 0,C 180,E1 1440.003,E2 1440.003} C_VEL
LIN {X 0,Y 592.267,Z 685.176,A -85,B 0,C 180,E1 1442.742,E2 1442.742} C_VEL
LIN {X 0,Y 592.356,Z 667.106,A -85,B 0,C 180,E1 1445.119,E2 1445.119} C_VEL
LIN {X 0,Y 592.551,Z 643.779,A -85,B 0,C 180,E1 1447.182,E2 1447.182} C_VEL
LIN {X 0,Y 592.693,Z 616.951,A -85,B 0,C 180,E1 1448.744,E2 1448.744} C_VEL
LIN {X 0,Y 592.908,Z 588.866,A -85,B 0,C 180,E1 1449.711,E2 1449.711} C_VEL
LIN {X 0,Y 591.854,Z 549.53,A -85,B 0,C 180,E1 1450.406,E2 1450.406} C_VEL
LIN {X 0,Y 591.616,Z 549.53,A -85,B 0,C 180,E1 1454.781,E2 1454.781} C_VEL
LIN {X 0,Y 591.736,Z 549.53,A -85,B 0,C 180,E1 1459.365,E2 1459.365} C_VEL
LIN {X 0,Y 591.633,Z 549.53,A -85,B 0,C 180,E1 1464.089,E2 1464.089} C_VEL
LIN {X 0,Y 591.628,Z 549.53,A -85,B 0,C 180,E1 1468.991,E2 1468.991} C_VEL
LIN {X 0,Y 591.705,Z 549.53,A -85,B 0,C 180,E1 1474.134,E2 1474.134} C_VEL
LIN {X 0,Y 591.523,Z 549.53,A -85,B 0,C 180,E1 1480.058,E2 1480.058} C_VEL
LIN {X 0,Y 591.608,Z 549.53,A -85,B 0,C 180,E1 1485.583,E2 1485.583} C_VEL
LIN {X 0,Y 591.571,Z 549.53,A -85,B 0,C 180,E1 1490.374,E2 1490.374} C_VEL
LIN {X 0,Y 591.628,Z 549.53,A -85,B 0,C 180,E1 1494.712,E2 1494.712} C_VEL
LIN {X 0,Y 591.554,Z 549.53,A -85,B 0,C 180,E1 1501.006,E2 1501.006} C_VEL
LIN {X 0,Y 591.954,Z 549.53,A -85,B 0,C 180,E1 1506.604,E2 1506.604} C_VEL
LIN {X 0,Y 591.995,Z 549.53,A -85,B 0,C 180,E1 1507.234,E2 1507.234} C_VEL
LIN {X 0,Y 594.118,Z 559.994,A -85,B 0,C 180,E1 1507.518,E2 1507.518} C_VEL
LIN {X 0,Y 593.854,Z 598.46,A -85,B 0,C 180,E1 1508.489,E2 1508.489} C_VEL
LIN {X 0,Y 593.505,Z 634.46,A -85,B 0,C 180,E1 1510.025,E2 1510.025} C_VEL
LIN {X 0,Y 593.114,Z 668.414,A -85,B 0,C 180,E1 1512.126,E2 1512.126} C_VEL
LIN {X 0,Y 592.686,Z 698.628,A -85,B 0,C 180,E1 1514.682,E2 1514.682} C_VEL
LIN {X 0,Y 592.316,Z 725.034,A -85,B 0,C 180,E1 1517.679,E2 1517.679} C_VEL
LIN {X 0,Y 592.121,Z 745.617,A -85,B 0,C 180,E1 1520.834,E2 1520.834} C_VEL
LIN {X 0,Y 592.016,Z 761.072,A -85,B 0,C 180,E1 1524.148,E2 1524.148} C_VEL
LIN {X 0,Y 592.065,Z 770.253,A -85,B 0,C 180,E1 1527.078,E2 1527.078} C_VEL
LIN {X 0,Y 592.062,Z 775.644,A -85,B 0,C 180,E1 1530,E2 1530} C_VEL
LIN {X 0,Y 592.026,Z 777.498,A -85,B 0,C 180,E1 1532.923,E2 1532.923} C_VEL
LIN {X 0,Y 592.052,Z 775.267,A -85,B 0,C 180,E1 1536.23,E2 1536.23} C_VEL
LIN {X 0,Y 592.128,Z 767.331,A -85,B 0,C 180,E1 1539.907,E2 1539.907} C_VEL
LIN {X 0,Y 592.15,Z 754.747,A -85,B 0,C 180,E1 1543.261,E2 1543.261} C_VEL
LIN {X 0,Y 592.28,Z 736.927,A -85,B 0,C 180,E1 1546.522,E2 1546.522} C_VEL
LIN {X 0,Y 592.574,Z 713.791,A -85,B 0,C 180,E1 1549.614,E2 1549.614} C_VEL
LIN {X 0,Y 592.892,Z 685.301,A -85,B 0,C 180,E1 1552.447,E2 1552.447} C_VEL
LIN {X 0,Y 593.278,Z 653.041,A -85,B 0,C 180,E1 1554.825,E2 1554.825} C_VEL
LIN {X 0,Y 593.748,Z 617.158,A -85,B 0,C 180,E1 1556.704,E2 1556.704} C_VEL
LIN {X 0,Y 594.008,Z 581.035,A -85,B 0,C 180,E1 1557.939,E2 1557.939} C_VEL
LIN {X 0,Y 593.353,Z 555.88,A -85,B 0,C 180,E1 1558.493,E2 1558.493} C_VEL
LIN {X 0,Y 591.558,Z 549.53,A -85,B 0,C 180,E1 1558.7,E2 1558.7} C_VEL
LIN {X 0,Y 591.9,Z 549.53,A -85,B 0,C 180,E1 1564.121,E2 1564.121} C_VEL
LIN {X 0,Y 591.588,Z 549.53,A -85,B 0,C 180,E1 1570.066,E2 1570.066} C_VEL
LIN {X 0,Y 591.416,Z 549.53,A -85,B 0,C 180,E1 1575.603,E2 1575.603} C_VEL
LIN {X 0,Y 591.588,Z 549.53,A -85,B 0,C 180,E1 1580.375,E2 1580.375} C_VEL
LIN {X 0,Y 591.876,Z 549.53,A -85,B 0,C 180,E1 1585.878,E2 1585.878} C_VEL
LIN {X 0,Y 591.682,Z 549.53,A -85,B 0,C 180,E1 1591.011,E2 1591.011} C_VEL
LIN {X 0,Y 591.691,Z 549.53,A -85,B 0,C 180,E1 1597.504,E2 1597.504} C_VEL
LIN {X 0,Y 591.497,Z 549.53,A -85,B 0,C 180,E1 1602.547,E2 1602.547} C_VEL
LIN {X 0,Y 590.864,Z 549.53,A -85,B 0,C 180,E1 1602.756,E2 1602.756} C_VEL
LIN {X 0,Y 592.72,Z 577.451,A -85,B 0,C 180,E1 1603.144,E2 1603.144} C_VEL
LIN {X 0,Y 592.685,Z 611.459,A -85,B 0,C 180,E1 1603.697,E2 1603.697} C_VEL
LIN {X 0,Y 592.514,Z 636.945,A -85,B 0,C 180,E1 1604.675,E2 1604.675} C_VEL
LIN {X 0,Y 592.384,Z 659.212,A -85,B 0,C 180,E1 1606.108,E2 1606.108} C_VEL
LIN {X 0,Y 592.216,Z 678.941,A -85,B 0,C 180,E1 1608.048,E2 1608.048} C_VEL
LIN {X 0,Y 592.145,Z 692.604,A -85,B 0,C 180,E1 1610.091,E2 1610.091} C_VEL
LIN {X 0,Y 592.129,Z 703.021,A -85,B 0,C 180,E1 1612.676,E2 1612.676} C_VEL
LIN {X 0,Y 592.181,Z 706.141,A -85,B 0,C 180,E1 1614.146,E2 1614.146} C_VEL
LIN {X 0,Y 592.058,Z 707.429,A -85,B 0,C 180,E1 1615.611,E2 1615.611} C_VEL
LIN {X 0,Y 592.085,Z 706.074,A -85,B 0,C 180,E1 1617.806,E2 1617.806} C_VEL
LIN {X 0,Y 592.132,Z 699.301,A -85,B 0,C 180,E1 1620.362,E2 1620.362} C_VEL
LIN {X 0,Y 592.244,Z 691.482,A -85,B 0,C 180,E1 1622.025,E2 1622.025} C_VEL
LIN {X 0,Y 588.221,Z 682.588,A -85,B 0,C 180,E1 1623.441,E2 1623.441} C_VEL
LIN {X 0,Y 584.473,Z 671.996,A -85,B 0,C 180,E1 1624.759,E2 1624.759} C_VEL
LIN {X 0,Y 584.677,Z 650.672,A -85,B 0,C 180,E1 1626.568,E2 1626.568} C_VEL
LIN {X 0,Y 584.875,Z 626.272,A -85,B 0,C 180,E1 1627.875,E2 1627.875} C_VEL
LIN {X 0,Y 585.042,Z 600.99,A -85,B 0,C 180,E1 1628.619,E2 1628.619} C_VEL
LIN {X 0,Y 584.232,Z 549.53,A -85,B 0,C 180,E1 1629.334,E2 1629.334} C_VEL
LIN {X 0,Y 583.859,Z 549.53,A -85,B 0,C 180,E1 1634.975,E2 1634.975} C_VEL
LIN {X 0,Y 583.798,Z 549.53,A -85,B 0,C 180,E1 1641.212,E2 1641.212} C_VEL
LIN {X 0,Y 583.717,Z 549.53,A -85,B 0,C 180,E1 1646.067,E2 1646.067} C_VEL
LIN {X 0,Y 583.592,Z 549.53,A -85,B 0,C 180,E1 1651.418,E2 1651.418} C_VEL
LIN {X 0,Y 583.738,Z 549.53,A -85,B 0,C 180,E1 1656.729,E2 1656.729} C_VEL
LIN {X 0,Y 583.753,Z 549.53,A -85,B 0,C 180,E1 1662.226,E2 1662.226} C_VEL
LIN {X 0,Y 583.544,Z 549.53,A -85,B 0,C 180,E1 1667.746,E2 1667.746} C_VEL
LIN {X 0,Y 583.511,Z 549.53,A -85,B 0,C 180,E1 1673.287,E2 1673.287} C_VEL
LIN {X 0,Y 583.876,Z 549.53,A -85,B 0,C 180,E1 1678.52,E2 1678.52} C_VEL
LIN {X 0,Y 583.925,Z 549.53,A -85,B 0,C 180,E1 1679.034,E2 1679.034} C_VEL
LIN {X 0,Y 587.753,Z 560.622,A -85,B 0,C 180,E1 1679.447,E2 1679.447} C_VEL
LIN {X 0,Y 587.768,Z 623.388,A -85,B 0,C 180,E1 1680.453,E2 1680.453} C_VEL
LIN {X 0,Y 587.306,Z 662.608,A -85,B 0,C 180,E1 1681.689,E2 1681.689} C_VEL
LIN {X 0,Y 586.64,Z 700.593,A -85,B 0,C 180,E1 1683.52,E2 1683.52} C_VEL
LIN {X 0,Y 585.898,Z 736.963,A -85,B 0,C 180,E1 1685.968,E2 1685.968} C_VEL
LIN {X 0,Y 585.258,Z 768.942,A -85,B 0,C 180,E1 1688.837,E2 1688.837} C_VEL
LIN {X 0,Y 584.748,Z 795.697,A -85,B 0,C 180,E1 1691.958,E2 1691.958} C_VEL
LIN {X 0,Y 584.366,Z 818.55,A -85,B 0,C 180,E1 1695.451,E2 1695.451} C_VEL
LIN {X 0,Y 584.227,Z 836.834,A -85,B 0,C 180,E1 1699.282,E2 1699.282} C_VEL
LIN {X 0,Y 584.153,Z 848.99,A -85,B 0,C 180,E1 1703.086,E2 1703.086} C_VEL
LIN {X 0,Y 584.082,Z 855.915,A -85,B 0,C 180,E1 1707.038,E2 1707.038} C_VEL
LIN {X 0,Y 584.049,Z 857.5,A -85,B 0,C 180,E1 1710,E2 1710} C_VEL
LIN {X 0,Y 584.026,Z 855.915,A -85,B 0,C 180,E1 1712.962,E2 1712.962} C_VEL
LIN {X 0,Y 584.084,Z 850.413,A -85,B 0,C 180,E1 1716.323,E2 1716.323} C_VEL
LIN {X 0,Y 584.07,Z 839.401,A -85,B 0,C 180,E1 1720.044,E2 1720.044} C_VEL
LIN {X 0,Y 584.312,Z 823.086,A -85,B 0,C 180,E1 1723.715,E2 1723.715} C_VEL
LIN {X 0,Y 584.618,Z 801.443,A -85,B 0,C 180,E1 1727.255,E2 1727.255} C_VEL
LIN {X 0,Y 585.109,Z 774.6,A -85,B 0,C 180,E1 1730.575,E2 1730.575} C_VEL
LIN {X 0,Y 585.776,Z 742.699,A -85,B 0,C 180,E1 1733.573,E2 1733.573} C_VEL
LIN {X 0,Y 586.441,Z 708.063,A -85,B 0,C 180,E1 1736.036,E2 1736.036} C_VEL
LIN {X 0,Y 587.147,Z 670.77,A -85,B 0,C 180,E1 1737.97,E2 1737.97} C_VEL
LIN {X 0,Y 587.663,Z 632.171,A -85,B 0,C 180,E1 1739.321,E2 1739.321} C_VEL
LIN {X 0,Y 587.975,Z 591.634,A -85,B 0,C 180,E1 1740.11,E2 1740.11} C_VEL
LIN {X 0,Y 587,Z 557.758,A -85,B 0,C 180,E1 1740.636,E2 1740.636} C_VEL
LIN {X 0,Y 583.839,Z 549.53,A -85,B 0,C 180,E1 1740.968,E2 1740.968} C_VEL
LIN {X 0,Y 583.829,Z 549.53,A -85,B 0,C 180,E1 1746.755,E2 1746.755} C_VEL
LIN {X 0,Y 583.57,Z 549.53,A -85,B 0,C 180,E1 1752.251,E2 1752.251} C_VEL
LIN {X 0,Y 583.741,Z 549.53,A -85,B 0,C 180,E1 1757.773,E2 1757.773} C_VEL
LIN {X 0,Y 583.755,Z 549.53,A -85,B 0,C 180,E1 1763.523,E2 1763.523} C_VEL
LIN {X 0,Y 583.663,Z 549.53,A -85,B 0,C 180,E1 1768.867,E2 1768.867} C_VEL
LIN {X 0,Y 583.824,Z 549.53,A -85,B 0,C 180,E1 1774.788,E2 1774.788} C_VEL
LIN {X 0,Y 584.003,Z 549.53,A -85,B 0,C 180,E1 1779.341,E2 1779.341} C_VEL
LIN {X 0,Y 585.189,Z 568.413,A -85,B 0,C 180,E1 1779.631,E2 1779.631} C_VEL
LIN {X 0,Y 585.221,Z 599.369,A -85,B 0,C 180,E1 1780.296,E2 1780.296} C_VEL
LIN {X 0,Y 584.974,Z 626.869,A -85,B 0,C 180,E1 1781.485,E2 1781.485} C_VEL
LIN {X 0,Y 584.646,Z 652.164,A -85,B 0,C 180,E1 1783.219,E2 1783.219} C_VEL
LIN {X 0,Y 584.434,Z 673.969,A -85,B 0,C 180,E1 1785.457,E2 1785.457} C_VEL
LIN {X 0,Y 584.289,Z 688.872,A -85,B 0,C 180,E1 1787.701,E2 1787.701} C_VEL
LIN {X 0,Y 584.195,Z 700.178,A -85,B 0,C 180,E1 1790.338,E2 1790.338} C_VEL
LIN {X 0,Y 584.233,Z 705.564,A -85,B 0,C 180,E1 1792.583,E2 1792.583} C_VEL
LIN {X 0,Y 584.19,Z 707.369,A -85,B 0,C 180,E1 1795.559,E2 1795.559} C_VEL
LIN {X 0,Y 584.249,Z 704.796,A -85,B 0,C 180,E1 1797.783,E2 1797.783} C_VEL
LIN {X 0,Y 584.286,Z 697.381,A -85,B 0,C 180,E1 1800.373,E2 1800.373} C_VEL
LIN {X 0,Y 584.387,Z 683.27,A -85,B 0,C 180,E1 1803.149,E2 1803.149} C_VEL
LIN {X 0,Y 584.55,Z 664.282,A -85,B 0,C 180,E1 1805.559,E2 1805.559} C_VEL
LIN {X 0,Y 584.804,Z 640.183,A -85,B 0,C 180,E1 1807.603,E2 1807.603} C_VEL
LIN {X 0,Y 585.054,Z 613.225,A -85,B 0,C 180,E1 1809.093,E2 1809.093} C_VEL
LIN {X 0,Y 585.348,Z 583.907,A -85,B 0,C 180,E1 1810.025,E2 1810.025} C_VEL
LIN {X 0,Y 583.974,Z 549.53,A -85,B 0,C 180,E1 1810.587,E2 1810.587} C_VEL
LIN {X 0,Y 583.709,Z 549.53,A -85,B 0,C 180,E1 1814.986,E2 1814.986} C_VEL
LIN {X 0,Y 583.794,Z 549.53,A -85,B 0,C 180,E1 1819.639,E2 1819.639} C_VEL
LIN {X 0,Y 583.673,Z 549.53,A -85,B 0,C 180,E1 1824.439,E2 1824.439} C_VEL
LIN {X 0,Y 583.637,Z 549.53,A -85,B 0,C 180,E1 1829.427,E2 1829.427} C_VEL
LIN {X 0,Y 583.687,Z 549.53,A -85,B 0,C 180,E1 1834.669,E2 1834.669} C_VEL
LIN {X 0,Y 583.588,Z 549.53,A -85,B 0,C 180,E1 1840.278,E2 1840.278} C_VEL
LIN {X 0,Y 583.719,Z 549.53,A -85,B 0,C 180,E1 1845.728,E2 1845.728} C_VEL
LIN {X 0,Y 583.703,Z 549.53,A -85,B 0,C 180,E1 1851.646,E2 1851.646} C_VEL
LIN {X 0,Y 583.501,Z 549.53,A -85,B 0,C 180,E1 1857.102,E2 1857.102} C_VEL
LIN {X 0,Y 583.609,Z 549.53,A -85,B 0,C 180,E1 1862.26,E2 1862.26} C_VEL
LIN {X 0,Y 584.065,Z 549.53,A -85,B 0,C 180,E1 1866.877,E2 1866.877} C_VEL
LIN {X 0,Y 587.012,Z 561.395,A -85,B 0,C 180,E1 1867.211,E2 1867.211} C_VEL
LIN {X 0,Y 586.596,Z 599.79,A -85,B 0,C 180,E1 1868.215,E2 1868.215} C_VEL
LIN {X 0,Y 586.129,Z 635.968,A -85,B 0,C 180,E1 1869.8,E2 1869.8} C_VEL
LIN {X 0,Y 585.557,Z 670.313,A -85,B 0,C 180,E1 1871.984,E2 1871.984} C_VEL
LIN {X 0,Y 585.008,Z 699.042,A -85,B 0,C 180,E1 1874.476,E2 1874.476} C_VEL
LIN {X 0,Y 584.554,Z 725.354,A -85,B 0,C 180,E1 1877.513,E2 1877.513} C_VEL
LIN {X 0,Y 584.293,Z 745.834,A -85,B 0,C 180,E1 1880.71,E2 1880.71} C_VEL
LIN {X 0,Y 584.14,Z 761.219,A -85,B 0,C 180,E1 1884.069,E2 1884.069} C_VEL
LIN {X 0,Y 584.187,Z 770.359,A -85,B 0,C 180,E1 1887.039,E2 1887.039} C_VEL
LIN {X 0,Y 584.171,Z 775.692,A -85,B 0,C 180,E1 1890,E2 1890} C_VEL
LIN {X 0,Y 584.141,Z 777.493,A -85,B 0,C 180,E1 1892.962,E2 1892.962} C_VEL
LIN {X 0,Y 584.146,Z 775.206,A -85,B 0,C 180,E1 1896.314,E2 1896.314} C_VEL
LIN {X 0,Y 584.241,Z 767.207,A -85,B 0,C 180,E1 1900.042,E2 1900.042} C_VEL
LIN {X 0,Y 584.303,Z 753.337,A -85,B 0,C 180,E1 1903.706,E2 1903.706} C_VEL
LIN {X 0,Y 584.494,Z 733.814,A -85,B 0,C 180,E1 1907.193,E2 1907.193} C_VEL
LIN {X 0,Y 584.862,Z 709.004,A -85,B 0,C 180,E1 1910.387,E2 1910.387} C_VEL
LIN {X 0,Y 585.359,Z 680.146,A -85,B 0,C 180,E1 1913.152,E2 1913.152} C_VEL
LIN {X 0,Y 585.954,Z 647.91,A -85,B 0,C 180,E1 1915.43,E2 1915.43} C_VEL
LIN {X 0,Y 586.48,Z 614.155,A -85,B 0,C 180,E1 1917.144,E2 1917.144} C_VEL
LIN {X 0,Y 586.888,Z 578.505,A -85,B 0,C 180,E1 1918.329,E2 1918.329} C_VEL
LIN {X 0,Y 586.121,Z 557.227,A -85,B 0,C 180,E1 1918.81,E2 1918.81} C_VEL
LIN {X 0,Y 583.617,Z 549.53,A -85,B 0,C 180,E1 1919.11,E2 1919.11} C_VEL
LIN {X 0,Y 583.916,Z 549.53,A -85,B 0,C 180,E1 1924.654,E2 1924.654} C_VEL
LIN {X 0,Y 583.668,Z 549.53,A -85,B 0,C 180,E1 1930.273,E2 1930.273} C_VEL
LIN {X 0,Y 583.607,Z 549.53,A -85,B 0,C 180,E1 1936.392,E2 1936.392} C_VEL
LIN {X 0,Y 583.75,Z 549.53,A -85,B 0,C 180,E1 1941.649,E2 1941.649} C_VEL
LIN {X 0,Y 583.879,Z 549.53,A -85,B 0,C 180,E1 1947.125,E2 1947.125} C_VEL
LIN {X 0,Y 583.645,Z 549.53,A -85,B 0,C 180,E1 1952.26,E2 1952.26} C_VEL
LIN {X 0,Y 583.767,Z 549.53,A -85,B 0,C 180,E1 1957.182,E2 1957.182} C_VEL
LIN {X 0,Y 583.336,Z 549.53,A -85,B 0,C 180,E1 1962.514,E2 1962.514} C_VEL
LIN {X 0,Y 585.02,Z 576.445,A -85,B 0,C 180,E1 1962.96,E2 1962.96} C_VEL
LIN {X 0,Y 584.984,Z 610.685,A -85,B 0,C 180,E1 1963.512,E2 1963.512} C_VEL
LIN {X 0,Y 584.799,Z 635.82,A -85,B 0,C 180,E1 1964.468,E2 1964.468} C_VEL
LIN {X 0,Y 584.566,Z 659.363,A -85,B 0,C 180,E1 1965.988,E2 1965.988} C_VEL
LIN {X 0,Y 584.377,Z 678.479,A -85,B 0,C 180,E1 1967.885,E2 1967.885} C_VEL
LIN {X 0,Y 584.284,Z 692.313,A -85,B 0,C 180,E1 1969.957,E2 1969.957} C_VEL
LIN {X 0,Y 584.231,Z 702.863,A -85,B 0,C 180,E1 1972.576,E2 1972.576} C_VEL
LIN {X 0,Y 584.281,Z 706.055,A -85,B 0,C 180,E1 1974.067,E2 1974.067} C_VEL
LIN {X 0,Y 584.166,Z 707.41,A -85,B 0,C 180,E1 1975.552,E2 1975.552} C_VEL
LIN {X 0,Y 584.211,Z 706.158,A -85,B 0,C 180,E1 1977.776,E2 1977.776} C_VEL
LIN {X 0,Y 584.236,Z 699.506,A -85,B 0,C 180,E1 1980.367,E2 1980.367} C_VEL
LIN {X 0,Y 584.335,Z 687.523,A -85,B 0,C 180,E1 1982.772,E2 1982.772} C_VEL
LIN {X 0,Y 584.473,Z 671.996,A -85,B 0,C 180,E1 1984.759,E2 1984.759} C_VEL
LIN {X 0,Y 582.052,Z 663.017,A -85,B 0,C 180,E1 1985.677,E2 1985.677} C_VEL
LIN {X 0,Y 576.953,Z 648.253,A -85,B 0,C 180,E1 1986.88,E2 1986.88} C_VEL
LIN {X 0,Y 576.906,Z 646.4,A -85,B 0,C 180,E1 1986.996,E2 1986.996} C_VEL
LIN {X 0,Y 577.204,Z 620.437,A -85,B 0,C 180,E1 1988.264,E2 1988.264} C_VEL
LIN {X 0,Y 577.359,Z 592.517,A -85,B 0,C 180,E1 1988.924,E2 1988.924} C_VEL
LIN {X 0,Y 576.326,Z 549.53,A -85,B 0,C 180,E1 1989.49,E2 1989.49} C_VEL
LIN {X 0,Y 575.94,Z 549.53,A -85,B 0,C 180,E1 1995.186,E2 1995.186} C_VEL
LIN {X 0,Y 575.83,Z 549.53,A -85,B 0,C 180,E1 2001.52,E2 2001.52} C_VEL
LIN {X 0,Y 575.661,Z 549.53,A -85,B 0,C 180,E1 2006.955,E2 2006.955} C_VEL
LIN {X 0,Y 575.682,Z 549.53,A -85,B 0,C 180,E1 2011.614,E2 2011.614} C_VEL
LIN {X 0,Y 575.824,Z 549.53,A -85,B 0,C 180,E1 2017.063,E2 2017.063} C_VEL
LIN {X 0,Y 575.817,Z 549.53,A -85,B 0,C 180,E1 2022.946,E2 2022.946} C_VEL
LIN {X 0,Y 575.653,Z 549.53,A -85,B 0,C 180,E1 2029.048,E2 2029.048} C_VEL
LIN {X 0,Y 575.707,Z 549.53,A -85,B 0,C 180,E1 2034.78,E2 2034.78} C_VEL
LIN {X 0,Y 576.017,Z 550.096,A -85,B 0,C 180,E1 2038.605,E2 2038.605} C_VEL
LIN {X 0,Y 580.953,Z 563.666,A -85,B 0,C 180,E1 2039.094,E2 2039.094} C_VEL
LIN {X 0,Y 580.909,Z 622.826,A -85,B 0,C 180,E1 2040.056,E2 2040.056} C_VEL
LIN {X 0,Y 580.345,Z 661.352,A -85,B 0,C 180,E1 2041.267,E2 2041.267} C_VEL
LIN {X 0,Y 579.49,Z 698.945,A -85,B 0,C 180,E1 2043.07,E2 2043.07} C_VEL
LIN {X 0,Y 578.52,Z 735.581,A -85,B 0,C 180,E1 2045.53,E2 2045.53} C_VEL
LIN {X 0,Y 577.693,Z 767.602,A -85,B 0,C 180,E1 2048.405,E2 2048.405} C_VEL
LIN {X 0,Y 577.016,Z 795.701,A -85,B 0,C 180,E1 2051.708,E2 2051.708} C_VEL
LIN {X 0,Y 576.555,Z 818.55,A -85,B 0,C 180,E1 2055.248,E2 2055.248} C_VEL
LIN {X 0,Y 576.348,Z 836.838,A -85,B 0,C 180,E1 2059.134,E2 2059.134} C_VEL
LIN {X 0,Y 576.213,Z 847.688,A -85,B 0,C 180,E1 2062.475,E2 2062.475} C_VEL
LIN {X 0,Y 576.096,Z 853.966,A -85,B 0,C 180,E1 2065.492,E2 2065.492} C_VEL
LIN {X 0,Y 576.133,Z 857.094,A -85,B 0,C 180,E1 2068.499,E2 2068.499} C_VEL
LIN {X 0,Y 576.28,Z 857.095,A -85,B 0,C 180,E1 2071.5,E2 2071.5} C_VEL
LIN {X 0,Y 576.256,Z 851.854,A -85,B 0,C 180,E1 2075.71,E2 2075.71} C_VEL
LIN {X 0,Y 576.279,Z 842.081,A -85,B 0,C 180,E1 2079.42,E2 2079.42} C_VEL
LIN {X 0,Y 576.465,Z 826.457,A -85,B 0,C 180,E1 2083.242,E2 2083.242} C_VEL
LIN {X 0,Y 576.774,Z 805.377,A -85,B 0,C 180,E1 2086.92,E2 2086.92} C_VEL
LIN {X 0,Y 577.372,Z 779.872,A -85,B 0,C 180,E1 2090.263,E2 2090.263} C_VEL
LIN {X 0,Y 578.125,Z 749.62,A -85,B 0,C 180,E1 2093.304,E2 2093.304} C_VEL
LIN {X 0,Y 579.025,Z 715.649,A -85,B 0,C 180,E1 2095.901,E2 2095.901} C_VEL
LIN {X 0,Y 579.923,Z 679.707,A -85,B 0,C 180,E1 2097.932,E2 2097.932} C_VEL
LIN {X 0,Y 580.613,Z 642.282,A -85,B 0,C 180,E1 2099.406,E2 2099.406} C_VEL
LIN {X 0,Y 581.169,Z 605.972,A -85,B 0,C 180,E1 2100.278,E2 2100.278} C_VEL
LIN {X 0,Y 580.29,Z 560.44,A -85,B 0,C 180,E1 2100.991,E2 2100.991} C_VEL
LIN {X 0,Y 575.854,Z 549.53,A -85,B 0,C 180,E1 2101.496,E2 2101.496} C_VEL
LIN {X 0,Y 575.92,Z 549.53,A -85,B 0,C 180,E1 2107.064,E2 2107.064} C_VEL
LIN {X 0,Y 575.68,Z 549.53,A -85,B 0,C 180,E1 2112.969,E2 2112.969} C_VEL
LIN {X 0,Y 575.814,Z 549.53,A -85,B 0,C 180,E1 2119.072,E2 2119.072} C_VEL
LIN {X 0,Y 575.712,Z 549.53,A -85,B 0,C 180,E1 2124.789,E2 2124.789} C_VEL
LIN {X 0,Y 575.741,Z 549.53,A -85,B 0,C 180,E1 2130.137,E2 2130.137} C_VEL
LIN {X 0,Y 575.887,Z 549.53,A -85,B 0,C 180,E1 2135.216,E2 2135.216} C_VEL
LIN {X 0,Y 576.035,Z 549.53,A -85,B 0,C 180,E1 2139.129,E2 2139.129} C_VEL
LIN {X 0,Y 577.481,Z 562.518,A -85,B 0,C 180,E1 2139.347,E2 2139.347} C_VEL
LIN {X 0,Y 577.573,Z 594.462,A -85,B 0,C 180,E1 2139.949,E2 2139.949} C_VEL
LIN {X 0,Y 577.273,Z 622.005,A -85,B 0,C 180,E1 2141.041,E2 2141.041} C_VEL
LIN {X 0,Y 576.94,Z 647.99,A -85,B 0,C 180,E1 2142.716,E2 2142.716} C_VEL
LIN {X 0,Y 576.657,Z 669.883,A -85,B 0,C 180,E1 2144.833,E2 2144.833} C_VEL
LIN {X 0,Y 576.45,Z 687.408,A -85,B 0,C 180,E1 2147.339,E2 2147.339} C_VEL
LIN {X 0,Y 576.337,Z 698.687,A -85,B 0,C 180,E1 2149.824,E2 2149.824} C_VEL
LIN {X 0,Y 576.336,Z 705.451,A -85,B 0,C 180,E1 2152.481,E2 2152.481} C_VEL
LIN {X 0,Y 576.285,Z 707.384,A -85,B 0,C 180,E1 2155.498,E2 2155.498} C_VEL
LIN {X 0,Y 576.359,Z 704.91,A -85,B 0,C 180,E1 2157.753,E2 2157.753} C_VEL
LIN {X 0,Y 576.39,Z 697.642,A -85,B 0,C 180,E1 2160.378,E2 2160.378} C_VEL
LIN {X 0,Y 576.509,Z 683.695,A -85,B 0,C 180,E1 2163.192,E2 2163.192} C_VEL
LIN {X 0,Y 576.715,Z 665.029,A -85,B 0,C 180,E1 2165.625,E2 2165.625} C_VEL
LIN {X 0,Y 577.038,Z 641.156,A -85,B 0,C 180,E1 2167.706,E2 2167.706} C_VEL
LIN {X 0,Y 577.376,Z 614.831,A -85,B 0,C 180,E1 2169.215,E2 2169.215} C_VEL
LIN {X 0,Y 577.713,Z 584.837,A -85,B 0,C 180,E1 2170.206,E2 2170.206} C_VEL
LIN {X 0,Y 576.456,Z 551.862,A -85,B 0,C 180,E1 2170.727,E2 2170.727} C_VEL
LIN {X 0,Y 576.101,Z 549.53,A -85,B 0,C 180,E1 2170.816,E2 2170.816} C_VEL
LIN {X 0,Y 575.986,Z 549.53,A -85,B 0,C 180,E1 2176.753,E2 2176.753} C_VEL
LIN {X 0,Y 575.871,Z 549.53,A -85,B 0,C 180,E1 2181.526,E2 2181.526} C_VEL
LIN {X 0,Y 575.789,Z 549.53,A -85,B 0,C 180,E1 2186.981,E2 2186.981} C_VEL
LIN {X 0,Y 575.844,Z 549.53,A -85,B 0,C 180,E1 2193.393,E2 2193.393} C_VEL
LIN {X 0,Y 575.668,Z 549.53,A -85,B 0,C 180,E1 2198.99,E2 2198.99} C_VEL
LIN {X 0,Y 575.776,Z 549.53,A -85,B 0,C 180,E1 2205.047,E2 2205.047} C_VEL
LIN {X 0,Y 575.744,Z 549.53,A -85,B 0,C 180,E1 2211.016,E2 2211.016} C_VEL
LIN {X 0,Y 575.594,Z 549.53,A -85,B 0,C 180,E1 2216.591,E2 2216.591} C_VEL
LIN {X 0,Y 575.698,Z 549.53,A -85,B 0,C 180,E1 2221.845,E2 2221.845} C_VEL
LIN {X 0,Y 576.168,Z 549.53,A -85,B 0,C 180,E1 2226.496,E2 2226.496} C_VEL
LIN {X 0,Y 579.905,Z 562.647,A -85,B 0,C 180,E1 2226.893,E2 2226.893} C_VEL
LIN {X 0,Y 579.395,Z 600.255,A -85,B 0,C 180,E1 2227.904,E2 2227.904} C_VEL
LIN {X 0,Y 578.823,Z 634.773,A -85,B 0,C 180,E1 2229.425,E2 2229.425} C_VEL
LIN {X 0,Y 578.059,Z 668.241,A -85,B 0,C 180,E1 2231.546,E2 2231.546} C_VEL
LIN {X 0,Y 577.396,Z 697.575,A -85,B 0,C 180,E1 2234.071,E2 2234.071} C_VEL
LIN {X 0,Y 576.81,Z 724.229,A -85,B 0,C 180,E1 2237.15,E2 2237.15} C_VEL
LIN {X 0,Y 576.491,Z 745.031,A -85,B 0,C 180,E1 2240.393,E2 2240.393} C_VEL
LIN {X 0,Y 576.271,Z 761.365,A -85,B 0,C 180,E1 2243.987,E2 2243.987} C_VEL
LIN {X 0,Y 576.293,Z 770.466,A -85,B 0,C 180,E1 2246.998,E2 2246.998} C_VEL
LIN {X 0,Y 576.27,Z 775.739,A -85,B 0,C 180,E1 2250,E2 2250} C_VEL
LIN {X 0,Y 576.236,Z 777.483,A -85,B 0,C 180,E1 2253.003,E2 2253.003} C_VEL
LIN {X 0,Y 576.251,Z 774.605,A -85,B 0,C 180,E1 2256.769,E2 2256.769} C_VEL
LIN {X 0,Y 576.335,Z 765.932,A -85,B 0,C 180,E1 2260.562,E2 2260.562} C_VEL
LIN {X 0,Y 576.426,Z 752.663,A -85,B 0,C 180,E1 2264.003,E2 2264.003} C_VEL
LIN {X 0,Y 576.68,Z 733.523,A -85,B 0,C 180,E1 2267.434,E2 2267.434} C_VEL
LIN {X 0,Y 577.183,Z 708.616,A -85,B 0,C 180,E1 2270.671,E2 2270.671} C_VEL
LIN {X 0,Y 577.818,Z 679.167,A -85,B 0,C 180,E1 2273.512,E2 2273.512} C_VEL
LIN {X 0,Y 578.575,Z 646.134,A -85,B 0,C 180,E1 2275.841,E2 2275.841} C_VEL
LIN {X 0,Y 579.277,Z 611.257,A -85,B 0,C 180,E1 2277.589,E2 2277.589} C_VEL
LIN {X 0,Y 579.832,Z 573.285,A -85,B 0,C 180,E1 2278.796,E2 2278.796} C_VEL
LIN {X 0,Y 579.018,Z 559.48,A -85,B 0,C 180,E1 2279.114,E2 2279.114} C_VEL
LIN {X 0,Y 575.714,Z 549.53,A -85,B 0,C 180,E1 2279.48,E2 2279.48} C_VEL
LIN {X 0,Y 576.015,Z 549.53,A -85,B 0,C 180,E1 2283.382,E2 2283.382} C_VEL
LIN {X 0,Y 575.765,Z 549.53,A -85,B 0,C 180,E1 2288.983,E2 2288.983} C_VEL
LIN {X 0,Y 575.717,Z 549.53,A -85,B 0,C 180,E1 2292.966,E2 2292.966} C_VEL
LIN {X 0,Y 575.781,Z 549.53,A -85,B 0,C 180,E1 2299.06,E2 2299.06} C_VEL
LIN {X 0,Y 575.933,Z 549.53,A -85,B 0,C 180,E1 2304.796,E2 2304.796} C_VEL
LIN {X 0,Y 575.795,Z 549.53,A -85,B 0,C 180,E1 2310.132,E2 2310.132} C_VEL
LIN {X 0,Y 575.765,Z 549.53,A -85,B 0,C 180,E1 2316.551,E2 2316.551} C_VEL
LIN {X 0,Y 575.544,Z 549.53,A -85,B 0,C 180,E1 2322.387,E2 2322.387} C_VEL
LIN {X 0,Y 577.314,Z 578.497,A -85,B 0,C 180,E1 2322.809,E2 2322.809} C_VEL
LIN {X 0,Y 577.249,Z 612.014,A -85,B 0,C 180,E1 2323.382,E2 2323.382} C_VEL
LIN {X 0,Y 576.995,Z 638.471,A -85,B 0,C 180,E1 2324.447,E2 2324.447} C_VEL
LIN {X 0,Y 576.757,Z 661.604,A -85,B 0,C 180,E1 2326.042,E2 2326.042} C_VEL
LIN {X 0,Y 576.505,Z 679.551,A -85,B 0,C 180,E1 2327.909,E2 2327.909} C_VEL
LIN {X 0,Y 576.38,Z 693.946,A -85,B 0,C 180,E1 2330.198,E2 2330.198} C_VEL
LIN {X 0,Y 576.343,Z 702.866,A -85,B 0,C 180,E1 2332.547,E2 2332.547} C_VEL
LIN {X 0,Y 576.345,Z 706.385,A -85,B 0,C 180,E1 2334.296,E2 2334.296} C_VEL
LIN {X 0,Y 576.307,Z 707.072,A -85,B 0,C 180,E1 2336.995,E2 2336.995} C_VEL
LIN {X 0,Y 576.389,Z 702.132,A -85,B 0,C 180,E1 2339.622,E2 2339.622} C_VEL
LIN {X 0,Y 576.438,Z 691.175,A -85,B 0,C 180,E1 2342.247,E2 2342.247} C_VEL
LIN {X 0,Y 576.611,Z 675.379,A -85,B 0,C 180,E1 2344.5,E2 2344.5} C_VEL
LIN {X 0,Y 576.838,Z 654.664,A -85,B 0,C 180,E1 2346.427,E2 2346.427} C_VEL
LIN {X 0,Y 576.906,Z 646.4,A -85,B 0,C 180,E1 2346.996,E2 2346.996} C_VEL
LIN {X 0,Y 574.631,Z 635.346,A -85,B 0,C 180,E1 2347.676,E2 2347.676} C_VEL
LIN {X 0,Y 569.759,Z 620.218,A -85,B 0,C 180,E1 2348.437,E2 2348.437} C_VEL
LIN {X 0,Y 569.517,Z 616.088,A -85,B 0,C 180,E1 2348.578,E2 2348.578} C_VEL
LIN {X 0,Y 569.664,Z 589.417,A -85,B 0,C 180,E1 2349.142,E2 2349.142} C_VEL
LIN {X 0,Y 568.711,Z 551.645,A -85,B 0,C 180,E1 2349.645,E2 2349.645} C_VEL
LIN {X 0,Y 568.41,Z 549.53,A -85,B 0,C 180,E1 2349.726,E2 2349.726} C_VEL
LIN {X 0,Y 568.008,Z 549.53,A -85,B 0,C 180,E1 2355.403,E2 2355.403} C_VEL
LIN {X 0,Y 567.94,Z 549.53,A -85,B 0,C 180,E1 2361.557,E2 2361.557} C_VEL
LIN {X 0,Y 567.771,Z 549.53,A -85,B 0,C 180,E1 2366.857,E2 2366.857} C_VEL
LIN {X 0,Y 567.706,Z 549.53,A -85,B 0,C 180,E1 2372.111,E2 2372.111} C_VEL
LIN {X 0,Y 567.901,Z 549.53,A -85,B 0,C 180,E1 2377.669,E2 2377.669} C_VEL
LIN {X 0,Y 567.815,Z 549.53,A -85,B 0,C 180,E1 2383.703,E2 2383.703} C_VEL
LIN {X 0,Y 567.686,Z 549.53,A -85,B 0,C 180,E1 2388.347,E2 2388.347} C_VEL
LIN {X 0,Y 567.736,Z 549.53,A -85,B 0,C 180,E1 2394.21,E2 2394.21} C_VEL
LIN {X 0,Y 568.083,Z 550.099,A -85,B 0,C 180,E1 2398.116,E2 2398.116} C_VEL
LIN {X 0,Y 574.146,Z 564.257,A -85,B 0,C 180,E1 2398.695,E2 2398.695} C_VEL
LIN {X 0,Y 574.004,Z 624.484,A -85,B 0,C 180,E1 2399.699,E2 2399.699} C_VEL
LIN {X 0,Y 573.256,Z 663.707,A -85,B 0,C 180,E1 2400.977,E2 2400.977} C_VEL
LIN {X 0,Y 572.262,Z 700.678,A -85,B 0,C 180,E1 2402.807,E2 2402.807} C_VEL
LIN {X 0,Y 571.12,Z 736.824,A -85,B 0,C 180,E1 2405.293,E2 2405.293} C_VEL
LIN {X 0,Y 570.087,Z 768.95,A -85,B 0,C 180,E1 2408.246,E2 2408.246} C_VEL
LIN {X 0,Y 569.285,Z 796.935,A -85,B 0,C 180,E1 2411.618,E2 2411.618} C_VEL
LIN {X 0,Y 568.736,Z 820.207,A -85,B 0,C 180,E1 2415.34,E2 2415.34} C_VEL
LIN {X 0,Y 568.494,Z 838.036,A -85,B 0,C 180,E1 2419.29,E2 2419.29} C_VEL
LIN {X 0,Y 568.366,Z 849.604,A -85,B 0,C 180,E1 2423.137,E2 2423.137} C_VEL
LIN {X 0,Y 568.267,Z 855.921,A -85,B 0,C 180,E1 2426.955,E2 2426.955} C_VEL
LIN {X 0,Y 568.267,Z 857.5,A -85,B 0,C 180,E1 2430,E2 2430} C_VEL
LIN {X 0,Y 568.226,Z 855.921,A -85,B 0,C 180,E1 2433.045,E2 2433.045} C_VEL
LIN {X 0,Y 568.293,Z 849.606,A -85,B 0,C 180,E1 2436.863,E2 2436.863} C_VEL
LIN {X 0,Y 568.387,Z 837.673,A -85,B 0,C 180,E1 2440.807,E2 2440.807} C_VEL
LIN {X 0,Y 568.739,Z 820.26,A -85,B 0,C 180,E1 2444.65,E2 2444.65} C_VEL
LIN {X 0,Y 569.295,Z 796.958,A -85,B 0,C 180,E1 2448.378,E2 2448.378} C_VEL
LIN {X 0,Y 570.097,Z 768.956,A -85,B 0,C 180,E1 2451.753,E2 2451.753} C_VEL
LIN {X 0,Y 571.062,Z 736.849,A -85,B 0,C 180,E1 2454.707,E2 2454.707} C_VEL
LIN {X 0,Y 572.221,Z 700.482,A -85,B 0,C 180,E1 2457.207,E2 2457.207} C_VEL
LIN {X 0,Y 573.247,Z 661.815,A -85,B 0,C 180,E1 2459.103,E2 2459.103} C_VEL
LIN {X 0,Y 574.031,Z 621.233,A -85,B 0,C 180,E1 2460.38,E2 2460.38} C_VEL
LIN {X 0,Y 573.66,Z 563.09,A -85,B 0,C 180,E1 2461.352,E2 2461.352} C_VEL
LIN {X 0,Y 567.869,Z 549.53,A -85,B 0,C 180,E1 2461.987,E2 2461.987} C_VEL
LIN {X 0,Y 567.999,Z 549.53,A -85,B 0,C 180,E1 2467.67,E2 2467.67} C_VEL
LIN {X 0,Y 567.74,Z 549.53,A -85,B 0,C 180,E1 2474.144,E2 2474.144} C_VEL
LIN {X 0,Y 567.843,Z 549.53,A -85,B 0,C 180,E1 2478.371,E2 2478.371} C_VEL
LIN {X 0,Y 567.854,Z 549.53,A -85,B 0,C 180,E1 2484.227,E2 2484.227} C_VEL
LIN {X 0,Y 567.832,Z 549.53,A -85,B 0,C 180,E1 2489.677,E2 2489.677} C_VEL
LIN {X 0,Y 567.933,Z 549.53,A -85,B 0,C 180,E1 2494.845,E2 2494.845} C_VEL
LIN {X 0,Y 568.116,Z 549.53,A -85,B 0,C 180,E1 2498.908,E2 2498.908} C_VEL
LIN {X 0,Y 569.902,Z 563.586,A -85,B 0,C 180,E1 2499.147,E2 2499.147} C_VEL
LIN {X 0,Y 569.908,Z 595.892,A -85,B 0,C 180,E1 2499.785,E2 2499.785} C_VEL
LIN {X 0,Y 569.541,Z 623.503,A -85,B 0,C 180,E1 2500.931,E2 2500.931} C_VEL
LIN {X 0,Y 569.136,Z 649.551,A -85,B 0,C 180,E1 2502.671,E2 2502.671} C_VEL
LIN {X 0,Y 568.803,Z 670.82,A -85,B 0,C 180,E1 2504.808,E2 2504.808} C_VEL
LIN {X 0,Y 568.589,Z 688.104,A -85,B 0,C 180,E1 2507.356,E2 2507.356} C_VEL
LIN {X 0,Y 568.457,Z 699.717,A -85,B 0,C 180,E1 2510.067,E2 2510.067} C_VEL
LIN {X 0,Y 568.433,Z 705.338,A -85,B 0,C 180,E1 2512.376,E2 2512.376} C_VEL
LIN {X 0,Y 568.394,Z 707.398,A -85,B 0,C 180,E1 2515.435,E2 2515.435} C_VEL
LIN {X 0,Y 568.483,Z 705.016,A -85,B 0,C 180,E1 2517.722,E2 2517.722} C_VEL
LIN {X 0,Y 568.494,Z 697.888,A -85,B 0,C 180,E1 2520.384,E2 2520.384} C_VEL
LIN {X 0,Y 568.649,Z 684.113,A -85,B 0,C 180,E1 2523.236,E2 2523.236} C_VEL
LIN {X 0,Y 568.876,Z 665.976,A -85,B 0,C 180,E1 2525.67,E2 2525.67} C_VEL
LIN {X 0,Y 569.281,Z 643.378,A -85,B 0,C 180,E1 2527.716,E2 2527.716} C_VEL
LIN {X 0,Y 569.596,Z 618.369,A -85,B 0,C 180,E1 2529.246,E2 2529.246} C_VEL
LIN {X 0,Y 570.035,Z 589.571,A -85,B 0,C 180,E1 2530.297,E2 2530.297} C_VEL
LIN {X 0,Y 569.008,Z 553.753,A -85,B 0,C 180,E1 2530.914,E2 2530.914} C_VEL
LIN {X 0,Y 568.225,Z 549.53,A -85,B 0,C 180,E1 2531.048,E2 2531.048} C_VEL
LIN {X 0,Y 568.067,Z 549.53,A -85,B 0,C 180,E1 2536.994,E2 2536.994} C_VEL
LIN {X 0,Y 567.953,Z 549.53,A -85,B 0,C 180,E1 2541.841,E2 2541.841} C_VEL
LIN {X 0,Y 567.876,Z 549.53,A -85,B 0,C 180,E1 2546.86,E2 2546.86} C_VEL
LIN {X 0,Y 567.847,Z 549.53,A -85,B 0,C 180,E1 2552.11,E2 2552.11} C_VEL
LIN {X 0,Y 567.679,Z 549.53,A -85,B 0,C 180,E1 2557.695,E2 2557.695} C_VEL
LIN {X 0,Y 567.745,Z 549.53,A -85,B 0,C 180,E1 2563.719,E2 2563.719} C_VEL
LIN {X 0,Y 567.822,Z 549.53,A -85,B 0,C 180,E1 2568.359,E2 2568.359} C_VEL
LIN {X 0,Y 567.834,Z 549.53,A -85,B 0,C 180,E1 2574.218,E2 2574.218} C_VEL
LIN {X 0,Y 567.802,Z 549.53,A -85,B 0,C 180,E1 2579.668,E2 2579.668} C_VEL
LIN {X 0,Y 568.245,Z 549.781,A -85,B 0,C 180,E1 2586.104,E2 2586.104} C_VEL
LIN {X 0,Y 572.816,Z 564.238,A -85,B 0,C 180,E1 2586.576,E2 2586.576} C_VEL
LIN {X 0,Y 572.154,Z 601.466,A -85,B 0,C 180,E1 2587.61,E2 2587.61} C_VEL
LIN {X 0,Y 571.416,Z 637.209,A -85,B 0,C 180,E1 2589.235,E2 2589.235} C_VEL
LIN {X 0,Y 570.494,Z 671.457,A -85,B 0,C 180,E1 2591.492,E2 2591.492} C_VEL
LIN {X 0,Y 569.628,Z 701.747,A -85,B 0,C 180,E1 2594.243,E2 2594.243} C_VEL
LIN {X 0,Y 568.98,Z 727.354,A -85,B 0,C 180,E1 2597.36,E2 2597.36} C_VEL
LIN {X 0,Y 568.654,Z 746.267,A -85,B 0,C 180,E1 2600.452,E2 2600.452} C_VEL
LIN {X 0,Y 568.39,Z 761.512,A -85,B 0,C 180,E1 2603.904,E2 2603.904} C_VEL
LIN {X 0,Y 568.399,Z 770.572,A -85,B 0,C 180,E1 2606.956,E2 2606.956} C_VEL
LIN {X 0,Y 568.384,Z 775.787,A -85,B 0,C 180,E1 2610,E2 2610} C_VEL
LIN {X 0,Y 568.33,Z 777.472,A -85,B 0,C 180,E1 2613.045,E2 2613.045} C_VEL
LIN {X 0,Y 568.357,Z 774.543,A -85,B 0,C 180,E1 2616.863,E2 2616.863} C_VEL
LIN {X 0,Y 568.423,Z 765.574,A -85,B 0,C 180,E1 2620.789,E2 2620.789} C_VEL
LIN {X 0,Y 568.551,Z 750.695,A -85,B 0,C 180,E1 2624.58,E2 2624.58} C_VEL
LIN {X 0,Y 568.894,Z 730.968,A -85,B 0,C 180,E1 2628.023,E2 2628.023} C_VEL
LIN {X 0,Y 569.552,Z 706.432,A -85,B 0,C 180,E1 2631.164,E2 2631.164} C_VEL
LIN {X 0,Y 570.343,Z 677.315,A -85,B 0,C 180,E1 2633.947,E2 2633.947} C_VEL
LIN {X 0,Y 571.238,Z 644.074,A -85,B 0,C 180,E1 2636.278,E2 2636.278} C_VEL
LIN {X 0,Y 572.085,Z 610.173,A -85,B 0,C 180,E1 2637.966,E2 2637.966} C_VEL
LIN {X 0,Y 572.712,Z 574.255,A -85,B 0,C 180,E1 2639.118,E2 2639.118} C_VEL
LIN {X 0,Y 571.849,Z 561.275,A -85,B 0,C 180,E1 2639.438,E2 2639.438} C_VEL
LIN {X 0,Y 567.785,Z 549.53,A -85,B 0,C 180,E1 2639.838,E2 2639.838} C_VEL
LIN {X 0,Y 567.985,Z 549.53,A -85,B 0,C 180,E1 2644.546,E2 2644.546} C_VEL
LIN {X 0,Y 567.828,Z 549.53,A -85,B 0,C 180,E1 2649.634,E2 2649.634} C_VEL
LIN {X 0,Y 567.664,Z 549.53,A -85,B 0,C 180,E1 2655.875,E2 2655.875} C_VEL
LIN {X 0,Y 567.84,Z 549.53,A -85,B 0,C 180,E1 2660.422,E2 2660.422} C_VEL
LIN {X 0,Y 568.015,Z 549.53,A -85,B 0,C 180,E1 2666.085,E2 2666.085} C_VEL
LIN {X 0,Y 567.824,Z 549.53,A -85,B 0,C 180,E1 2671.418,E2 2671.418} C_VEL
LIN {X 0,Y 567.867,Z 549.53,A -85,B 0,C 180,E1 2676.505,E2 2676.505} C_VEL
LIN {X 0,Y 567.763,Z 549.53,A -85,B 0,C 180,E1 2682.204,E2 2682.204} C_VEL
LIN {X 0,Y 569.649,Z 577.915,A -85,B 0,C 180,E1 2682.622,E2 2682.622} C_VEL
LIN {X 0,Y 569.538,Z 611.683,A -85,B 0,C 180,E1 2683.2,E2 2683.2} C_VEL
LIN {X 0,Y 569.279,Z 637.377,A -85,B 0,C 180,E1 2684.231,E2 2684.231} C_VEL
LIN {X 0,Y 568.942,Z 660.433,A -85,B 0,C 180,E1 2685.805,E2 2685.805} C_VEL
LIN {X 0,Y 568.661,Z 679.11,A -85,B 0,C 180,E1 2687.74,E2 2687.74} C_VEL
LIN {X 0,Y 568.512,Z 693.658,A -85,B 0,C 180,E1 2690.061,E2 2690.061} C_VEL
LIN {X 0,Y 568.446,Z 702.94,A -85,B 0,C 180,E1 2692.541,E2 2692.541} C_VEL
LIN {X 0,Y 568.479,Z 705.883,A -85,B 0,C 180,E1 2693.901,E2 2693.901} C_VEL
LIN {X 0,Y 568.379,Z 707.344,A -85,B 0,C 180,E1 2695.428,E2 2695.428} C_VEL
LIN {X 0,Y 568.448,Z 706.281,A -85,B 0,C 180,E1 2697.714,E2 2697.714} C_VEL
LIN {X 0,Y 568.446,Z 699.909,A -85,B 0,C 180,E1 2700.377,E2 2700.377} C_VEL
LIN {X 0,Y 568.583,Z 687.042,A -85,B 0,C 180,E1 2703.039,E2 2703.039} C_VEL
LIN {X 0,Y 568.804,Z 670.125,A -85,B 0,C 180,E1 2705.196,E2 2705.196} C_VEL
LIN {X 0,Y 569.132,Z 648.102,A -85,B 0,C 180,E1 2707.04,E2 2707.04} C_VEL
LIN {X 0,Y 569.464,Z 623.062,A -85,B 0,C 180,E1 2708.329,E2 2708.329} C_VEL
LIN {X 0,Y 569.517,Z 616.088,A -85,B 0,C 180,E1 2708.578,E2 2708.578} C_VEL
LIN {X 0,Y 567.444,Z 603.682,A -85,B 0,C 180,E1 2708.964,E2 2708.964} C_VEL
LIN {X 0,Y 562.049,Z 585.061,A -85,B 0,C 180,E1 2709.38,E2 2709.38} C_VEL
LIN {X 0,Y 561.944,Z 582.89,A -85,B 0,C 180,E1 2709.41,E2 2709.41} C_VEL
LIN {X 0,Y 560.955,Z 552.125,A -85,B 0,C 180,E1 2709.832,E2 2709.832} C_VEL
LIN {X 0,Y 560.491,Z 549.53,A -85,B 0,C 180,E1 2709.884,E2 2709.884} C_VEL
LIN {X 0,Y 560.078,Z 549.53,A -85,B 0,C 180,E1 2715.627,E2 2715.627} C_VEL
LIN {X 0,Y 560.032,Z 549.53,A -85,B 0,C 180,E1 2720.501,E2 2720.501} C_VEL
LIN {X 0,Y 559.914,Z 549.53,A -85,B 0,C 180,E1 2725.541,E2 2725.541} C_VEL
LIN {X 0,Y 559.842,Z 549.53,A -85,B 0,C 180,E1 2730.802,E2 2730.802} C_VEL
LIN {X 0,Y 559.945,Z 549.53,A -85,B 0,C 180,E1 2736.358,E2 2736.358} C_VEL
LIN {X 0,Y 559.91,Z 549.53,A -85,B 0,C 180,E1 2742.355,E2 2742.355} C_VEL
LIN {X 0,Y 559.767,Z 549.53,A -85,B 0,C 180,E1 2747.621,E2 2747.621} C_VEL
LIN {X 0,Y 559.809,Z 549.53,A -85,B 0,C 180,E1 2753.962,E2 2753.962} C_VEL
LIN {X 0,Y 560.12,Z 550.148,A -85,B 0,C 180,E1 2757.608,E2 2757.608} C_VEL
LIN {X 0,Y 567.417,Z 566.783,A -85,B 0,C 180,E1 2758.317,E2 2758.317} C_VEL
LIN {X 0,Y 567.166,Z 624.475,A -85,B 0,C 180,E1 2759.295,E2 2759.295} C_VEL
LIN {X 0,Y 566.313,Z 663.144,A -85,B 0,C 180,E1 2760.563,E2 2760.563} C_VEL
LIN {X 0,Y 565.1,Z 700.538,A -85,B 0,C 180,E1 2762.425,E2 2762.425} C_VEL
LIN {X 0,Y 563.775,Z 736.539,A -85,B 0,C 180,E1 2764.926,E2 2764.926} C_VEL
LIN {X 0,Y 562.528,Z 768.954,A -85,B 0,C 180,E1 2767.938,E2 2767.938} C_VEL
LIN {X 0,Y 561.578,Z 796.804,A -85,B 0,C 180,E1 2771.338,E2 2771.338} C_VEL
LIN {X 0,Y 560.929,Z 819.79,A -85,B 0,C 180,E1 2775.053,E2 2775.053} C_VEL
LIN {X 0,Y 560.632,Z 838.035,A -85,B 0,C 180,E1 2779.138,E2 2779.138} C_VEL
LIN {X 0,Y 560.479,Z 849.604,A -85,B 0,C 180,E1 2783.04,E2 2783.04} C_VEL
LIN {X 0,Y 560.361,Z 855.924,A -85,B 0,C 180,E1 2786.912,E2 2786.912} C_VEL
LIN {X 0,Y 560.368,Z 857.5,A -85,B 0,C 180,E1 2790,E2 2790} C_VEL
LIN {X 0,Y 560.325,Z 855.924,A -85,B 0,C 180,E1 2793.088,E2 2793.088} C_VEL
LIN {X 0,Y 560.424,Z 849.605,A -85,B 0,C 180,E1 2796.96,E2 2796.96} C_VEL
LIN {X 0,Y 560.514,Z 838.038,A -85,B 0,C 180,E1 2800.863,E2 2800.863} C_VEL
LIN {X 0,Y 560.945,Z 820.253,A -85,B 0,C 180,E1 2804.859,E2 2804.859} C_VEL
LIN {X 0,Y 561.599,Z 797.178,A -85,B 0,C 180,E1 2808.609,E2 2808.609} C_VEL
LIN {X 0,Y 562.485,Z 770.871,A -85,B 0,C 180,E1 2811.856,E2 2811.856} C_VEL
LIN {X 0,Y 563.607,Z 739.969,A -85,B 0,C 180,E1 2814.793,E2 2814.793} C_VEL
LIN {X 0,Y 564.837,Z 705.72,A -85,B 0,C 180,E1 2817.263,E2 2817.263} C_VEL
LIN {X 0,Y 566.097,Z 668.083,A -85,B 0,C 180,E1 2819.232,E2 2819.232} C_VEL
LIN {X 0,Y 566.96,Z 629.21,A -85,B 0,C 180,E1 2820.588,E2 2820.588} C_VEL
LIN {X 0,Y 567.524,Z 582.736,A -85,B 0,C 180,E1 2821.444,E2 2821.444} C_VEL
LIN {X 0,Y 566.722,Z 565.298,A -85,B 0,C 180,E1 2821.748,E2 2821.748} C_VEL
LIN {X 0,Y 559.885,Z 549.53,A -85,B 0,C 180,E1 2822.455,E2 2822.455} C_VEL
LIN {X 0,Y 559.986,Z 549.53,A -85,B 0,C 180,E1 2828.305,E2 2828.305} C_VEL
LIN {X 0,Y 559.811,Z 549.53,A -85,B 0,C 180,E1 2834.501,E2 2834.501} C_VEL
LIN {X 0,Y 559.867,Z 549.53,A -85,B 0,C 180,E1 2839.698,E2 2839.698} C_VEL
LIN {X 0,Y 559.839,Z 549.53,A -85,B 0,C 180,E1 2845.529,E2 2845.529} C_VEL
LIN {X 0,Y 559.865,Z 549.53,A -85,B 0,C 180,E1 2850.981,E2 2850.981} C_VEL
LIN {X 0,Y 559.943,Z 549.53,A -85,B 0,C 180,E1 2856.402,E2 2856.402} C_VEL
LIN {X 0,Y 560.138,Z 549.712,A -85,B 0,C 180,E1 2858.683,E2 2858.683} C_VEL
LIN {X 0,Y 562.313,Z 563.945,A -85,B 0,C 180,E1 2858.933,E2 2858.933} C_VEL
LIN {X 0,Y 562.313,Z 594.869,A -85,B 0,C 180,E1 2859.545,E2 2859.545} C_VEL
LIN {X 0,Y 561.894,Z 622.193,A -85,B 0,C 180,E1 2860.665,E2 2860.665} C_VEL
LIN {X 0,Y 561.416,Z 648.643,A -85,B 0,C 180,E1 2862.425,E2 2862.425} C_VEL
LIN {X 0,Y 560.999,Z 670.053,A -85,B 0,C 180,E1 2864.571,E2 2864.571} C_VEL
LIN {X 0,Y 560.755,Z 687.698,A -85,B 0,C 180,E1 2867.176,E2 2867.176} C_VEL
LIN {X 0,Y 560.575,Z 699.529,A -85,B 0,C 180,E1 2869.94,E2 2869.94} C_VEL
LIN {X 0,Y 560.539,Z 705.224,A -85,B 0,C 180,E1 2872.268,E2 2872.268} C_VEL
LIN {X 0,Y 560.487,Z 707.412,A -85,B 0,C 180,E1 2875.371,E2 2875.371} C_VEL
LIN {X 0,Y 560.604,Z 705.123,A -85,B 0,C 180,E1 2877.689,E2 2877.689} C_VEL
LIN {X 0,Y 560.611,Z 698.133,A -85,B 0,C 180,E1 2880.389,E2 2880.389} C_VEL
LIN {X 0,Y 560.783,Z 684.531,A -85,B 0,C 180,E1 2883.282,E2 2883.282} C_VEL
LIN {X 0,Y 561.061,Z 666.241,A -85,B 0,C 180,E1 2885.791,E2 2885.791} C_VEL
LIN {X 0,Y 561.516,Z 643.028,A -85,B 0,C 180,E1 2887.92,E2 2887.92} C_VEL
LIN {X 0,Y 561.939,Z 618.115,A -85,B 0,C 180,E1 2889.458,E2 2889.458} C_VEL
LIN {X 0,Y 562.403,Z 590.015,A -85,B 0,C 180,E1 2890.498,E2 2890.498} C_VEL
LIN {X 0,Y 561.492,Z 555.186,A -85,B 0,C 180,E1 2891.115,E2 2891.115} C_VEL
LIN {X 0,Y 560.324,Z 549.53,A -85,B 0,C 180,E1 2891.244,E2 2891.244} C_VEL
LIN {X 0,Y 560.142,Z 549.53,A -85,B 0,C 180,E1 2897.242,E2 2897.242} C_VEL
LIN {X 0,Y 560.011,Z 549.53,A -85,B 0,C 180,E1 2902.167,E2 2902.167} C_VEL
LIN {X 0,Y 559.951,Z 549.53,A -85,B 0,C 180,E1 2907.271,E2 2907.271} C_VEL
LIN {X 0,Y 559.89,Z 549.53,A -85,B 0,C 180,E1 2913.322,E2 2913.322} C_VEL
LIN {X 0,Y 559.736,Z 549.53,A -85,B 0,C 180,E1 2918.565,E2 2918.565} C_VEL
LIN {X 0,Y 559.828,Z 549.53,A -85,B 0,C 180,E1 2924.499,E2 2924.499} C_VEL
LIN {X 0,Y 559.845,Z 549.53,A -85,B 0,C 180,E1 2929.687,E2 2929.687} C_VEL
LIN {X 0,Y 559.809,Z 549.53,A -85,B 0,C 180,E1 2935.519,E2 2935.519} C_VEL
LIN {X 0,Y 559.845,Z 549.53,A -85,B 0,C 180,E1 2940.973,E2 2940.973} C_VEL
LIN {X 0,Y 560.308,Z 549.53,A -85,B 0,C 180,E1 2945.679,E2 2945.679} C_VEL
LIN {X 0,Y 565.718,Z 565.968,A -85,B 0,C 180,E1 2946.257,E2 2946.257} C_VEL
LIN {X 0,Y 564.938,Z 603.857,A -85,B 0,C 180,E1 2947.354,E2 2947.354} C_VEL
LIN {X 0,Y 564.025,Z 639.363,A -85,B 0,C 180,E1 2949.031,E2 2949.031} C_VEL
LIN {X 0,Y 562.943,Z 673.301,A -85,B 0,C 180,E1 2951.34,E2 2951.34} C_VEL
LIN {X 0,Y 561.98,Z 702.153,A -85,B 0,C 180,E1 2954.023,E2 2954.023} C_VEL
LIN {X 0,Y 561.193,Z 727.642,A -85,B 0,C 180,E1 2957.182,E2 2957.182} C_VEL
LIN {X 0,Y 560.743,Z 748.457,A -85,B 0,C 180,E1 2960.707,E2 2960.707} C_VEL
LIN {X 0,Y 560.502,Z 762.971,A -85,B 0,C 180,E1 2964.201,E2 2964.201} C_VEL
LIN {X 0,Y 560.486,Z 772.269,A -85,B 0,C 180,E1 2967.686,E2 2967.686} C_VEL
LIN {X 0,Y 560.384,Z 777.115,A -85,B 0,C 180,E1 2971.544,E2 2971.544} C_VEL
LIN {X 0,Y 560.412,Z 776.762,A -85,B 0,C 180,E1 2974.887,E2 2974.887} C_VEL
LIN {X 0,Y 560.444,Z 771.687,A -85,B 0,C 180,E1 2978.517,E2 2978.517} C_VEL
LIN {X 0,Y 560.496,Z 761.831,A -85,B 0,C 180,E1 2982.045,E2 2982.045} C_VEL
LIN {X 0,Y 560.826,Z 745.382,A -85,B 0,C 180,E1 2985.811,E2 2985.811} C_VEL
LIN {X 0,Y 561.366,Z 723.293,A -85,B 0,C 180,E1 2989.334,E2 2989.334} C_VEL
LIN {X 0,Y 562.139,Z 698.028,A -85,B 0,C 180,E1 2992.326,E2 2992.326} C_VEL
LIN {X 0,Y 563.141,Z 666.921,A -85,B 0,C 180,E1 2995.066,E2 2995.066} C_VEL
LIN {X 0,Y 564.142,Z 633.723,A -85,B 0,C 180,E1 2997.19,E2 2997.19} C_VEL
LIN {X 0,Y 565.105,Z 597.643,A -85,B 0,C 180,E1 2998.787,E2 2998.787} C_VEL
LIN {X 0,Y 565.007,Z 564.101,A -85,B 0,C 180,E1 2999.727,E2 2999.727} C_VEL
LIN {X 0,Y 559.909,Z 549.53,A -85,B 0,C 180,E1 3000.32,E2 3000.32} C_VEL
LIN {X 0,Y 560.062,Z 549.53,A -85,B 0,C 180,E1 3006.062,E2 3006.062} C_VEL
LIN {X 0,Y 559.825,Z 549.53,A -85,B 0,C 180,E1 3012.373,E2 3012.373} C_VEL
LIN {X 0,Y 559.84,Z 549.53,A -85,B 0,C 180,E1 3017.629,E2 3017.629} C_VEL
LIN {X 0,Y 560.097,Z 549.53,A -85,B 0,C 180,E1 3023.935,E2 3023.935} C_VEL
LIN {X 0,Y 560.007,Z 549.53,A -85,B 0,C 180,E1 3029.585,E2 3029.585} C_VEL
LIN {X 0,Y 559.907,Z 549.53,A -85,B 0,C 180,E1 3036.151,E2 3036.151} C_VEL
LIN {X 0,Y 559.99,Z 549.53,A -85,B 0,C 180,E1 3042.019,E2 3042.019} C_VEL
LIN {X 0,Y 561.965,Z 576.802,A -85,B 0,C 180,E1 3042.422,E2 3042.422} C_VEL
LIN {X 0,Y 561.83,Z 611.352,A -85,B 0,C 180,E1 3043.013,E2 3043.013} C_VEL
LIN {X 0,Y 561.519,Z 638.144,A -85,B 0,C 180,E1 3044.107,E2 3044.107} C_VEL
LIN {X 0,Y 561.108,Z 660.408,A -85,B 0,C 180,E1 3045.661,E2 3045.661} C_VEL
LIN {X 0,Y 560.8,Z 680.159,A -85,B 0,C 180,E1 3047.762,E2 3047.762} C_VEL
LIN {X 0,Y 560.629,Z 695.244,A -85,B 0,C 180,E1 3050.312,E2 3050.312} C_VEL
LIN {X 0,Y 560.563,Z 704.288,A -85,B 0,C 180,E1 3053.039,E2 3053.039} C_VEL
LIN {X 0,Y 560.486,Z 707.312,A -85,B 0,C 180,E1 3055.364,E2 3055.364} C_VEL
LIN {X 0,Y 560.57,Z 706.341,A -85,B 0,C 180,E1 3057.682,E2 3057.682} C_VEL
LIN {X 0,Y 560.565,Z 700.107,A -85,B 0,C 180,E1 3060.382,E2 3060.382} C_VEL
LIN {X 0,Y 560.703,Z 687.381,A -85,B 0,C 180,E1 3063.082,E2 3063.082} C_VEL
LIN {X 0,Y 560.979,Z 670.18,A -85,B 0,C 180,E1 3065.319,E2 3065.319} C_VEL
LIN {X 0,Y 561.342,Z 648.931,A -85,B 0,C 180,E1 3067.139,E2 3067.139} C_VEL
LIN {X 0,Y 561.716,Z 624.464,A -85,B 0,C 180,E1 3068.445,E2 3068.445} C_VEL
LIN {X 0,Y 561.982,Z 599.748,A -85,B 0,C 180,E1 3069.17,E2 3069.17} C_VEL
LIN {X 0,Y 561.944,Z 582.89,A -85,B 0,C 180,E1 3069.41,E2 3069.41} C_VEL
LIN {X 0,Y 558.137,Z 571.935,A -85,B 0,C 180,E1 3069.646,E2 3069.646} C_VEL
LIN {X 0,Y 554.193,Z 560.986,A -85,B 0,C 180,E1 3069.888,E2 3069.888} C_VEL
LIN {X 0,Y 552.542,Z 549.53,A -85,B 0,C 180,E1 3070.123,E2 3070.123} C_VEL
LIN {X 0,Y 552.115,Z 549.53,A -85,B 0,C 180,E1 3076.92,E2 3076.92} C_VEL
LIN {X 0,Y 552.007,Z 549.53,A -85,B 0,C 180,E1 3082.498,E2 3082.498} C_VEL
LIN {X 0,Y 551.878,Z 549.53,A -85,B 0,C 180,E1 3087.696,E2 3087.696} C_VEL
LIN {X 0,Y 551.826,Z 549.53,A -85,B 0,C 180,E1 3093.152,E2 3093.152} C_VEL
LIN {X 0,Y 551.974,Z 549.53,A -85,B 0,C 180,E1 3098.956,E2 3098.956} C_VEL
LIN {X 0,Y 551.936,Z 549.53,A -85,B 0,C 180,E1 3104.689,E2 3104.689} C_VEL
LIN {X 0,Y 551.846,Z 549.53,A -85,B 0,C 180,E1 3109.96,E2 3109.96} C_VEL
LIN {X 0,Y 551.988,Z 549.53,A -85,B 0,C 180,E1 3115.093,E2 3115.093} C_VEL
LIN {X 0,Y 552.126,Z 549.642,A -85,B 0,C 180,E1 3117.073,E2 3117.073} C_VEL
LIN {X 0,Y 560.712,Z 569.978,A -85,B 0,C 180,E1 3117.941,E2 3117.941} C_VEL
LIN {X 0,Y 560.344,Z 625.162,A -85,B 0,C 180,E1 3118.898,E2 3118.898} C_VEL
LIN {X 0,Y 559.35,Z 663.469,A -85,B 0,C 180,E1 3120.174,E2 3120.174} C_VEL
LIN {X 0,Y 557.944,Z 701.203,A -85,B 0,C 180,E1 3122.082,E2 3122.082} C_VEL
LIN {X 0,Y 556.373,Z 737.404,A -85,B 0,C 180,E1 3124.642,E2 3124.642} C_VEL
LIN {X 0,Y 554.98,Z 768.958,A -85,B 0,C 180,E1 3127.622,E2 3127.622} C_VEL
LIN {X 0,Y 553.866,Z 795.714,A -85,B 0,C 180,E1 3130.914,E2 3130.914} C_VEL
LIN {X 0,Y 553.091,Z 817.806,A -85,B 0,C 180,E1 3134.467,E2 3134.467} C_VEL
LIN {X 0,Y 552.671,Z 834.997,A -85,B 0,C 180,E1 3138.182,E2 3138.182} C_VEL
LIN {X 0,Y 552.534,Z 847.698,A -85,B 0,C 180,E1 3142.15,E2 3142.15} C_VEL
LIN {X 0,Y 552.461,Z 853.974,A -85,B 0,C 180,E1 3145.299,E2 3145.299} C_VEL
LIN {X 0,Y 552.46,Z 857.101,A -85,B 0,C 180,E1 3148.434,E2 3148.434} C_VEL
LIN {X 0,Y 552.583,Z 857.101,A -85,B 0,C 180,E1 3151.565,E2 3151.565} C_VEL
LIN {X 0,Y 552.547,Z 852.377,A -85,B 0,C 180,E1 3155.695,E2 3155.695} C_VEL
LIN {X 0,Y 552.613,Z 843.319,A -85,B 0,C 180,E1 3159.431,E2 3159.431} C_VEL
LIN {X 0,Y 552.925,Z 828.294,A -85,B 0,C 180,E1 3163.415,E2 3163.415} C_VEL
LIN {X 0,Y 553.48,Z 806.932,A -85,B 0,C 180,E1 3167.41,E2 3167.41} C_VEL
LIN {X 0,Y 554.448,Z 781.614,A -85,B 0,C 180,E1 3170.931,E2 3170.931} C_VEL
LIN {X 0,Y 555.793,Z 750.989,A -85,B 0,C 180,E1 3174.172,E2 3174.172} C_VEL
LIN {X 0,Y 557.222,Z 716.708,A -85,B 0,C 180,E1 3176.919,E2 3176.919} C_VEL
LIN {X 0,Y 558.72,Z 681.665,A -85,B 0,C 180,E1 3178.989,E2 3178.989} C_VEL
LIN {X 0,Y 559.891,Z 644.839,A -85,B 0,C 180,E1 3180.521,E2 3180.521} C_VEL
LIN {X 0,Y 560.761,Z 607.568,A -85,B 0,C 180,E1 3181.477,E2 3181.477} C_VEL
LIN {X 0,Y 560.125,Z 568.012,A -85,B 0,C 180,E1 3182.126,E2 3182.126} C_VEL
LIN {X 0,Y 551.945,Z 549.53,A -85,B 0,C 180,E1 3183.01,E2 3183.01} C_VEL
LIN {X 0,Y 552.013,Z 549.53,A -85,B 0,C 180,E1 3188.962,E2 3188.962} C_VEL
LIN {X 0,Y 551.935,Z 549.53,A -85,B 0,C 180,E1 3195.31,E2 3195.31} C_VEL
LIN {X 0,Y 551.979,Z 549.53,A -85,B 0,C 180,E1 3201.044,E2 3201.044} C_VEL
LIN {X 0,Y 551.886,Z 549.53,A -85,B 0,C 180,E1 3206.852,E2 3206.852} C_VEL
LIN {X 0,Y 551.961,Z 549.53,A -85,B 0,C 180,E1 3212.309,E2 3212.309} C_VEL
LIN {X 0,Y 552.223,Z 549.53,A -85,B 0,C 180,E1 3218.443,E2 3218.443} C_VEL
LIN {X 0,Y 554.731,Z 563.81,A -85,B 0,C 180,E1 3218.706,E2 3218.706} C_VEL
LIN {X 0,Y 554.685,Z 595.428,A -85,B 0,C 180,E1 3219.345,E2 3219.345} C_VEL
LIN {X 0,Y 554.197,Z 623.24,A -85,B 0,C 180,E1 3220.523,E2 3220.523} C_VEL
LIN {X 0,Y 553.64,Z 648.686,A -85,B 0,C 180,E1 3222.25,E2 3222.25} C_VEL
LIN {X 0,Y 553.172,Z 669.672,A -85,B 0,C 180,E1 3224.376,E2 3224.376} C_VEL
LIN {X 0,Y 552.913,Z 687.289,A -85,B 0,C 180,E1 3226.991,E2 3226.991} C_VEL
LIN {X 0,Y 552.721,Z 698.025,A -85,B 0,C 180,E1 3229.407,E2 3229.407} C_VEL
LIN {X 0,Y 552.638,Z 705.111,A -85,B 0,C 180,E1 3232.157,E2 3232.157} C_VEL
LIN {X 0,Y 552.606,Z 707.408,A -85,B 0,C 180,E1 3235.305,E2 3235.305} C_VEL
LIN {X 0,Y 552.707,Z 705.229,A -85,B 0,C 180,E1 3237.656,E2 3237.656} C_VEL
LIN {X 0,Y 552.729,Z 698.374,A -85,B 0,C 180,E1 3240.395,E2 3240.395} C_VEL
LIN {X 0,Y 552.897,Z 686.109,A -85,B 0,C 180,E1 3243.133,E2 3243.133} C_VEL
LIN {X 0,Y 553.214,Z 667.658,A -85,B 0,C 180,E1 3245.777,E2 3245.777} C_VEL
LIN {X 0,Y 553.751,Z 645.251,A -85,B 0,C 180,E1 3247.933,E2 3247.933} C_VEL
LIN {X 0,Y 554.227,Z 619.222,A -85,B 0,C 180,E1 3249.604,E2 3249.604} C_VEL
LIN {X 0,Y 554.786,Z 590.881,A -85,B 0,C 180,E1 3250.694,E2 3250.694} C_VEL
LIN {X 0,Y 554.069,Z 556.964,A -85,B 0,C 180,E1 3251.314,E2 3251.314} C_VEL
LIN {X 0,Y 552.446,Z 549.53,A -85,B 0,C 180,E1 3251.466,E2 3251.466} C_VEL
LIN {X 0,Y 552.224,Z 549.53,A -85,B 0,C 180,E1 3257.497,E2 3257.497} C_VEL
LIN {X 0,Y 552.078,Z 549.53,A -85,B 0,C 180,E1 3262.503,E2 3262.503} C_VEL
LIN {X 0,Y 551.992,Z 549.53,A -85,B 0,C 180,E1 3267.698,E2 3267.698} C_VEL
LIN {X 0,Y 551.982,Z 549.53,A -85,B 0,C 180,E1 3273.15,E2 3273.15} C_VEL
LIN {X 0,Y 551.802,Z 549.53,A -85,B 0,C 180,E1 3278.98,E2 3278.98} C_VEL
LIN {X 0,Y 551.934,Z 549.53,A -85,B 0,C 180,E1 3284.69,E2 3284.69} C_VEL
LIN {X 0,Y 551.938,Z 549.53,A -85,B 0,C 180,E1 3289.96,E2 3289.96} C_VEL
LIN {X 0,Y 551.904,Z 549.53,A -85,B 0,C 180,E1 3295.118,E2 3295.118} C_VEL
LIN {X 0,Y 551.952,Z 549.53,A -85,B 0,C 180,E1 3301.038,E2 3301.038} C_VEL
LIN {X 0,Y 552.35,Z 549.53,A -85,B 0,C 180,E1 3305.241,E2 3305.241} C_VEL
LIN {X 0,Y 558.653,Z 567.698,A -85,B 0,C 180,E1 3305.93,E2 3305.93} C_VEL
LIN {X 0,Y 557.729,Z 606.526,A -85,B 0,C 180,E1 3307.102,E2 3307.102} C_VEL
LIN {X 0,Y 556.619,Z 641.799,A -85,B 0,C 180,E1 3308.842,E2 3308.842} C_VEL
LIN {X 0,Y 555.411,Z 674.799,A -85,B 0,C 180,E1 3311.158,E2 3311.158} C_VEL
LIN {X 0,Y 554.264,Z 704.426,A -85,B 0,C 180,E1 3313.997,E2 3313.997} C_VEL
LIN {X 0,Y 553.392,Z 729.244,A -85,B 0,C 180,E1 3317.198,E2 3317.198} C_VEL
LIN {X 0,Y 552.92,Z 748.673,A -85,B 0,C 180,E1 3320.575,E2 3320.575} C_VEL
LIN {X 0,Y 552.613,Z 763.131,A -85,B 0,C 180,E1 3324.122,E2 3324.122} C_VEL
LIN {X 0,Y 552.598,Z 772.353,A -85,B 0,C 180,E1 3327.652,E2 3327.652} C_VEL
LIN {X 0,Y 552.49,Z 777.133,A -85,B 0,C 180,E1 3331.566,E2 3331.566} C_VEL
LIN {X 0,Y 552.55,Z 776.9,A -85,B 0,C 180,E1 3334.7,E2 3334.7} C_VEL
LIN {X 0,Y 552.545,Z 771.604,A -85,B 0,C 180,E1 3338.64,E2 3338.64} C_VEL
LIN {X 0,Y 552.631,Z 761.684,A -85,B 0,C 180,E1 3342.219,E2 3342.219} C_VEL
LIN {X 0,Y 552.959,Z 746.166,A -85,B 0,C 180,E1 3345.839,E2 3345.839} C_VEL
LIN {X 0,Y 553.534,Z 725.05,A -85,B 0,C 180,E1 3349.324,E2 3349.324} C_VEL
LIN {X 0,Y 554.46,Z 699.942,A -85,B 0,C 180,E1 3352.4,E2 3352.4} C_VEL
LIN {X 0,Y 555.59,Z 669.413,A -85,B 0,C 180,E1 3355.184,E2 3355.184} C_VEL
LIN {X 0,Y 556.776,Z 636.701,A -85,B 0,C 180,E1 3357.364,E2 3357.364} C_VEL
LIN {X 0,Y 557.885,Z 600.578,A -85,B 0,C 180,E1 3359.035,E2 3359.035} C_VEL
LIN {X 0,Y 557.906,Z 566.219,A -85,B 0,C 180,E1 3360.049,E2 3360.049} C_VEL
LIN {X 0,Y 552.034,Z 549.53,A -85,B 0,C 180,E1 3360.692,E2 3360.692} C_VEL
LIN {X 0,Y 552.148,Z 549.53,A -85,B 0,C 180,E1 3365.029,E2 3365.029} C_VEL
LIN {X 0,Y 551.965,Z 549.53,A -85,B 0,C 180,E1 3371.012,E2 3371.012} C_VEL
LIN {X 0,Y 551.934,Z 549.53,A -85,B 0,C 180,E1 3377.585,E2 3377.585} C_VEL
LIN {X 0,Y 552.075,Z 549.53,A -85,B 0,C 180,E1 3383.029,E2 3383.029} C_VEL
LIN {X 0,Y 552.055,Z 549.53,A -85,B 0,C 180,E1 3388.706,E2 3388.706} C_VEL
LIN {X 0,Y 551.884,Z 549.53,A -85,B 0,C 180,E1 3394.478,E2 3394.478} C_VEL
LIN {X 0,Y 551.886,Z 549.53,A -85,B 0,C 180,E1 3399.175,E2 3399.175} C_VEL
LIN {X 0,Y 552.13,Z 550.267,A -85,B 0,C 180,E1 3401.831,E2 3401.831} C_VEL
LIN {X 0,Y 554.295,Z 575.8,A -85,B 0,C 180,E1 3402.218,E2 3402.218} C_VEL
LIN {X 0,Y 554.144,Z 611.026,A -85,B 0,C 180,E1 3402.821,E2 3402.821} C_VEL
LIN {X 0,Y 553.803,Z 637.019,A -85,B 0,C 180,E1 3403.88,E2 3403.88} C_VEL
LIN {X 0,Y 553.346,Z 659.72,A -85,B 0,C 180,E1 3405.455,E2 3405.455} C_VEL
LIN {X 0,Y 552.954,Z 679.724,A -85,B 0,C 180,E1 3407.586,E2 3407.586} C_VEL
LIN {X 0,Y 552.779,Z 693.911,A -85,B 0,C 180,E1 3409.951,E2 3409.951} C_VEL
LIN {X 0,Y 552.673,Z 703.283,A -85,B 0,C 180,E1 3412.544,E2 3412.544} C_VEL
LIN {X 0,Y 552.605,Z 707.279,A -85,B 0,C 180,E1 3415.297,E2 3415.297} C_VEL
LIN {X 0,Y 552.617,Z 707.178,A -85,B 0,C 180,E1 3416.866,E2 3416.866} C_VEL
LIN {X 0,Y 552.727,Z 702.607,A -85,B 0,C 180,E1 3419.605,E2 3419.605} C_VEL
LIN {X 0,Y 552.797,Z 692.085,A -85,B 0,C 180,E1 3422.343,E2 3422.343} C_VEL
LIN {X 0,Y 553.051,Z 676.766,A -85,B 0,C 180,E1 3424.692,E2 3424.692} C_VEL
LIN {X 0,Y 553.441,Z 656.276,A -85,B 0,C 180,E1 3426.749,E2 3426.749} C_VEL
LIN {X 0,Y 553.874,Z 631.343,A -85,B 0,C 180,E1 3428.319,E2 3428.319} C_VEL
LIN {X 0,Y 554.228,Z 604.895,A -85,B 0,C 180,E1 3429.25,E2 3429.25} C_VEL
LIN {X 0,Y 554.193,Z 560.986,A -85,B 0,C 180,E1 3429.888,E2 3429.888} C_VEL
LIN {X 0,Y 552.309,Z 554.562,A -85,B 0,C 180,E1 3430.309,E2 3430.309} C_VEL
LIN {X 0,Y 548.149,Z 550.639,A -85,B 0,C 180,E1 3431.273,E2 3431.273} C_VEL
LIN {X 0,Y 544.332,Z 549.539,A -85,B 0,C 180,E1 3432.728,E2 3432.728} C_VEL
LIN {X 0,Y 544.209,Z 549.53,A -85,B 0,C 180,E1 3432.982,E2 3432.982} C_VEL
LIN {X 0,Y 544.182,Z 549.53,A -85,B 0,C 180,E1 3437.756,E2 3437.756} C_VEL
LIN {X 0,Y 544.033,Z 549.53,A -85,B 0,C 180,E1 3443.731,E2 3443.731} C_VEL
LIN {X 0,Y 543.94,Z 549.53,A -85,B 0,C 180,E1 3449.954,E2 3449.954} C_VEL
LIN {X 0,Y 544.01,Z 549.53,A -85,B 0,C 180,E1 3456.436,E2 3456.436} C_VEL
LIN {X 0,Y 544.073,Z 549.53,A -85,B 0,C 180,E1 3461.728,E2 3461.728} C_VEL
LIN {X 0,Y 543.944,Z 549.53,A -85,B 0,C 180,E1 3468.25,E2 3468.25} C_VEL
LIN {X 0,Y 543.952,Z 549.53,A -85,B 0,C 180,E1 3474.363,E2 3474.363} C_VEL
LIN {X 0,Y 544.165,Z 549.53,A -85,B 0,C 180,E1 3476.52,E2 3476.52} C_VEL
LIN {X 0,Y 554.027,Z 573.25,A -85,B 0,C 180,E1 3477.556,E2 3477.556} C_VEL
LIN {X 0,Y 553.562,Z 624.524,A -85,B 0,C 180,E1 3478.457,E2 3478.457} C_VEL
LIN {X 0,Y 552.449,Z 663.021,A -85,B 0,C 180,E1 3479.743,E2 3479.743} C_VEL
LIN {X 0,Y 550.889,Z 700.011,A -85,B 0,C 180,E1 3481.617,E2 3481.617} C_VEL
LIN {X 0,Y 549.107,Z 736.388,A -85,B 0,C 180,E1 3484.195,E2 3484.195} C_VEL
LIN {X 0,Y 547.434,Z 768.962,A -85,B 0,C 180,E1 3487.297,E2 3487.297} C_VEL
LIN {X 0,Y 546.171,Z 795.718,A -85,B 0,C 180,E1 3490.635,E2 3490.635} C_VEL
LIN {X 0,Y 545.282,Z 818.368,A -85,B 0,C 180,E1 3494.344,E2 3494.344} C_VEL
LIN {X 0,Y 544.83,Z 835,A -85,B 0,C 180,E1 3498.009,E2 3498.009} C_VEL
LIN {X 0,Y 544.712,Z 846.71,A -85,B 0,C 180,E1 3501.636,E2 3501.636} C_VEL
LIN {X 0,Y 544.56,Z 853.976,A -85,B 0,C 180,E1 3505.231,E2 3505.231} C_VEL
LIN {X 0,Y 544.558,Z 857.103,A -85,B 0,C 180,E1 3508.412,E2 3508.412} C_VEL
LIN {X 0,Y 544.677,Z 857.103,A -85,B 0,C 180,E1 3511.587,E2 3511.587} C_VEL
LIN {X 0,Y 544.658,Z 852.748,A -85,B 0,C 180,E1 3515.565,E2 3515.565} C_VEL
LIN {X 0,Y 544.715,Z 843.322,A -85,B 0,C 180,E1 3519.569,E2 3519.569} C_VEL
LIN {X 0,Y 545.09,Z 828.453,A -85,B 0,C 180,E1 3523.575,E2 3523.575} C_VEL
LIN {X 0,Y 545.726,Z 807.78,A -85,B 0,C 180,E1 3527.526,E2 3527.526} C_VEL
LIN {X 0,Y 546.849,Z 781.722,A -85,B 0,C 180,E1 3531.223,E2 3531.223} C_VEL
LIN {X 0,Y 548.366,Z 751.265,A -85,B 0,C 180,E1 3534.495,E2 3534.495} C_VEL
LIN {X 0,Y 549.976,Z 718.018,A -85,B 0,C 180,E1 3537.208,E2 3537.208} C_VEL
LIN {X 0,Y 551.699,Z 682.087,A -85,B 0,C 180,E1 3539.372,E2 3539.372} C_VEL
LIN {X 0,Y 553.043,Z 644.165,A -85,B 0,C 180,E1 3540.964,E2 3540.964} C_VEL
LIN {X 0,Y 554.052,Z 606.916,A -85,B 0,C 180,E1 3541.914,E2 3541.914} C_VEL
LIN {X 0,Y 553.471,Z 570.823,A -85,B 0,C 180,E1 3542.517,E2 3542.517} C_VEL
LIN {X 0,Y 544.018,Z 549.53,A -85,B 0,C 180,E1 3543.551,E2 3543.551} C_VEL
LIN {X 0,Y 544.098,Z 549.53,A -85,B 0,C 180,E1 3549.059,E2 3549.059} C_VEL
LIN {X 0,Y 543.95,Z 549.53,A -85,B 0,C 180,E1 3553.917,E2 3553.917} C_VEL
LIN {X 0,Y 544.07,Z 549.53,A -85,B 0,C 180,E1 3558.499,E2 3558.499} C_VEL
LIN {X 0,Y 543.991,Z 549.53,A -85,B 0,C 180,E1 3564.375,E2 3564.375} C_VEL
LIN {X 0,Y 543.999,Z 549.53,A -85,B 0,C 180,E1 3570.05,E2 3570.05} C_VEL
LIN {X 0,Y 544.107,Z 549.53,A -85,B 0,C 180,E1 3575.421,E2 3575.421} C_VEL
LIN {X 0,Y 544.265,Z 549.53,A -85,B 0,C 180,E1 3578.246,E2 3578.246} C_VEL
LIN {X 0,Y 547.083,Z 565.771,A -85,B 0,C 180,E1 3578.537,E2 3578.537} C_VEL
